RoboDK station: robodk_line_following_configuration_analysis.rdk

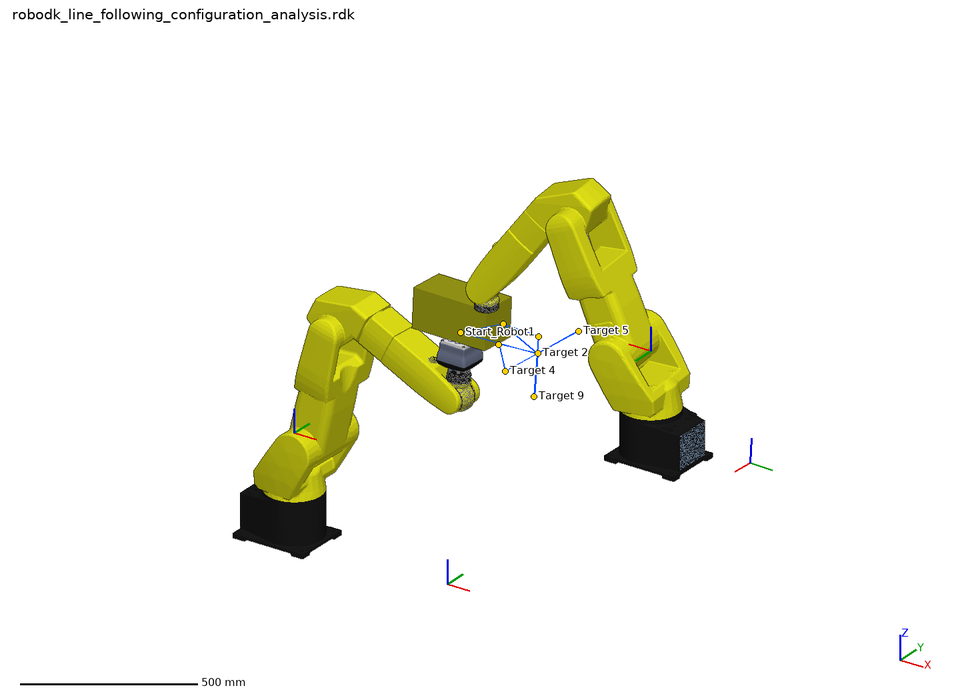
[picture v0: the station drawn from its stored meshes, robots at their saved joint values, targets as dots, program paths as lines]
Station Zavrsni_Line_Following_konfg (saved by RoboDK 5.9.4). Poses are relative to the parent item; angles as X-Y-Z fixed-axis rotations.
  - frame Pozicija 1 at (0, 0, 0) mm
    - frame Robot2 at (1093.21, 1000, 570) mm
      - robot Robot1: 6 axes
          modified DH rows (alpha deg, a mm, theta deg, d mm): 0, 0, 0, 330; -90, 75, -90, 0; 0, 400, 0, 0; -90, 75, 0, 410; 90, 0, 0, 0; -90, 0, 0, 80
          base shift (0, 0, -330) mm
          joint limits [-170, -60, -70, -190, -115, -400] to [170, 140, 170, 190, 115, 400]; home [0, 0, 0, 0, 0, 0]; saved at [-1.125, 13.477, -25.633, 3.463, 114.965, -89.87]
        - frame Kocka_Frame at (0, 1000, 0) mm
          - target Start_Robot2 (Cartesian target) at (63.45, -874.36, 243.45) mm, rotated rx 176.87 ry 0.69 rz -90 deg; joints [6.118, 22.277, -53.703, 0.008, -36.284, -5.881] of Robot2
          - target Kut_2 (Cartesian target) at (63.45, -1124.36, 243.45) mm, rotated rx 176.87 ry 0 rz -90 deg; joints [4.228, 52.378, -32.499, 0.062, -56.803, -4.056] of Robot2
          - target Kut_3 (Cartesian target) at (-60.55, -1124.36, 243.45) mm, rotated rx 176.87 ry 0 rz -90 deg; joints [-4.893, 52.997, -32.992, -0.071, -56.31, 5.138] of Robot2
          - target Kut_4 (Cartesian target) at (-60.55, -874.35, 243.45) mm, rotated rx 176.87 ry 0.69 rz -90.24 deg; joints [-7.279, 23.195, -54.517, 0, -35.483, 7.279] of Robot2
          - target Line_001 (Cartesian target) at (63.45, -874.36, 243.45) mm, rotated rx 176.87 ry 0.69 rz -90 deg; joints [-1.125, 13.477, -25.633, 3.463, 114.965, -89.87] of Robot2
          - target Line_002 (Cartesian target) at (63.45, -876.88, 243.45) mm, rotated rx 176.87 ry 0.69 rz -90 deg; joints [-1.125, 13.477, -25.633, 3.463, 114.965, -89.87] of Robot2
          - target Line_003 (Cartesian target) at (63.45, -879.41, 243.45) mm, rotated rx 176.87 ry 0.69 rz -90 deg; joints [-1.125, 13.477, -25.633, 3.463, 114.965, -89.87] of Robot2
          - target Line_004 (Cartesian target) at (63.45, -881.93, 243.45) mm, rotated rx 176.87 ry 0.69 rz -90 deg; joints [-1.125, 13.477, -25.633, 3.463, 114.965, -89.87] of Robot2
          - target Line_005 (Cartesian target) at (63.45, -884.46, 243.45) mm, rotated rx 176.87 ry 0.69 rz -90 deg; joints [-1.125, 13.477, -25.633, 3.463, 114.965, -89.87] of Robot2
          - target Line_006 (Cartesian target) at (63.45, -886.98, 243.45) mm, rotated rx 176.87 ry 0.69 rz -90 deg; joints [-1.125, 13.477, -25.633, 3.463, 114.965, -89.87] of Robot2
          - target Line_007 (Cartesian target) at (63.45, -889.51, 243.45) mm, rotated rx 176.87 ry 0.69 rz -90 deg; joints [-1.125, 13.477, -25.633, 3.463, 114.965, -89.87] of Robot2
          - target Line_008 (Cartesian target) at (63.45, -892.03, 243.45) mm, rotated rx 176.87 ry 0.69 rz -90 deg; joints [-1.125, 13.477, -25.633, 3.463, 114.965, -89.87] of Robot2
          - target Line_009 (Cartesian target) at (63.45, -894.56, 243.45) mm, rotated rx 176.87 ry 0.69 rz -90 deg; joints [-1.125, 13.477, -25.633, 3.463, 114.965, -89.87] of Robot2
          - target Line_010 (Cartesian target) at (63.45, -897.08, 243.45) mm, rotated rx 176.87 ry 0.69 rz -90 deg; joints [-1.125, 13.477, -25.633, 3.463, 114.965, -89.87] of Robot2
          - target Line_011 (Cartesian target) at (63.45, -899.61, 243.45) mm, rotated rx 176.87 ry 0.69 rz -90 deg; joints [-1.125, 13.477, -25.633, 3.463, 114.965, -89.87] of Robot2
          - target Line_012 (Cartesian target) at (63.45, -902.13, 243.45) mm, rotated rx 176.87 ry 0.69 rz -90 deg; joints [-1.125, 13.477, -25.633, 3.463, 114.965, -89.87] of Robot2
          - target Line_013 (Cartesian target) at (63.45, -904.66, 243.45) mm, rotated rx 176.87 ry 0.69 rz -90 deg; joints [-1.125, 13.477, -25.633, 3.463, 114.965, -89.87] of Robot2
          - target Line_014 (Cartesian target) at (63.45, -907.18, 243.45) mm, rotated rx 176.87 ry 0.69 rz -90 deg; joints [-1.125, 13.477, -25.633, 3.463, 114.965, -89.87] of Robot2
          - target Line_015 (Cartesian target) at (63.45, -909.71, 243.45) mm, rotated rx 176.87 ry 0.69 rz -90 deg; joints [-1.125, 13.477, -25.633, 3.463, 114.965, -89.87] of Robot2
          - target Line_016 (Cartesian target) at (63.45, -912.23, 243.45) mm, rotated rx 176.87 ry 0.69 rz -90 deg; joints [-1.125, 13.477, -25.633, 3.463, 114.965, -89.87] of Robot2
          - target Line_017 (Cartesian target) at (63.45, -914.76, 243.45) mm, rotated rx 176.87 ry 0.69 rz -90 deg; joints [-1.125, 13.477, -25.633, 3.463, 114.965, -89.87] of Robot2
          - target Line_018 (Cartesian target) at (63.45, -917.28, 243.45) mm, rotated rx 176.87 ry 0.69 rz -90 deg; joints [-1.125, 13.477, -25.633, 3.463, 114.965, -89.87] of Robot2
          - target Line_019 (Cartesian target) at (63.45, -919.81, 243.45) mm, rotated rx 176.87 ry 0.69 rz -90 deg; joints [-1.125, 13.477, -25.633, 3.463, 114.965, -89.87] of Robot2
          - target Line_020 (Cartesian target) at (63.45, -922.33, 243.45) mm, rotated rx 176.87 ry 0.69 rz -90 deg; joints [-1.125, 13.477, -25.633, 3.463, 114.965, -89.87] of Robot2
          - target Line_021 (Cartesian target) at (63.45, -924.86, 243.45) mm, rotated rx 176.87 ry 0.69 rz -90 deg; joints [-1.125, 13.477, -25.633, 3.463, 114.965, -89.87] of Robot2
          - target Line_022 (Cartesian target) at (63.45, -927.39, 243.45) mm, rotated rx 176.87 ry 0.69 rz -90 deg; joints [-1.125, 13.477, -25.633, 3.463, 114.965, -89.87] of Robot2
          - target Line_023 (Cartesian target) at (63.45, -929.91, 243.45) mm, rotated rx 176.87 ry 0.69 rz -90 deg; joints [-1.125, 13.477, -25.633, 3.463, 114.965, -89.87] of Robot2
          - target Line_024 (Cartesian target) at (63.45, -932.44, 243.45) mm, rotated rx 176.87 ry 0.69 rz -90 deg; joints [-1.125, 13.477, -25.633, 3.463, 114.965, -89.87] of Robot2
          - target Line_025 (Cartesian target) at (63.45, -934.96, 243.45) mm, rotated rx 176.87 ry 0.69 rz -90 deg; joints [-1.125, 13.477, -25.633, 3.463, 114.965, -89.87] of Robot2
          - target Line_026 (Cartesian target) at (63.45, -937.49, 243.45) mm, rotated rx 176.87 ry 0.69 rz -90 deg; joints [-1.125, 13.477, -25.633, 3.463, 114.965, -89.87] of Robot2
          - target Line_027 (Cartesian target) at (63.45, -940.01, 243.45) mm, rotated rx 176.87 ry 0.69 rz -90 deg; joints [-1.125, 13.477, -25.633, 3.463, 114.965, -89.87] of Robot2
          - target Line_028 (Cartesian target) at (63.45, -942.54, 243.45) mm, rotated rx 176.87 ry 0.69 rz -90 deg; joints [-1.125, 13.477, -25.633, 3.463, 114.965, -89.87] of Robot2
          - target Line_029 (Cartesian target) at (63.45, -945.06, 243.45) mm, rotated rx 176.87 ry 0.69 rz -90 deg; joints [-1.125, 13.477, -25.633, 3.463, 114.965, -89.87] of Robot2
          - target Line_030 (Cartesian target) at (63.45, -947.59, 243.45) mm, rotated rx 176.87 ry 0.69 rz -90 deg; joints [-1.125, 13.477, -25.633, 3.463, 114.965, -89.87] of Robot2
          - target Line_031 (Cartesian target) at (63.45, -950.11, 243.45) mm, rotated rx 176.87 ry 0.69 rz -90 deg; joints [-1.125, 13.477, -25.633, 3.463, 114.965, -89.87] of Robot2
          - target Line_032 (Cartesian target) at (63.45, -952.64, 243.45) mm, rotated rx 176.87 ry 0.69 rz -90 deg; joints [-1.125, 13.477, -25.633, 3.463, 114.965, -89.87] of Robot2
          - target Line_033 (Cartesian target) at (63.45, -955.16, 243.45) mm, rotated rx 176.87 ry 0.69 rz -90 deg; joints [-1.125, 13.477, -25.633, 3.463, 114.965, -89.87] of Robot2
          - target Line_034 (Cartesian target) at (63.45, -957.69, 243.45) mm, rotated rx 176.87 ry 0.69 rz -90 deg; joints [-1.125, 13.477, -25.633, 3.463, 114.965, -89.87] of Robot2
          - target Line_035 (Cartesian target) at (63.45, -960.21, 243.45) mm, rotated rx 176.87 ry 0.69 rz -90 deg; joints [-1.125, 13.477, -25.633, 3.463, 114.965, -89.87] of Robot2
          - target Line_036 (Cartesian target) at (63.45, -962.74, 243.45) mm, rotated rx 176.87 ry 0.69 rz -90 deg; joints [-1.125, 13.477, -25.633, 3.463, 114.965, -89.87] of Robot2
          - target Line_037 (Cartesian target) at (63.45, -965.26, 243.45) mm, rotated rx 176.87 ry 0.69 rz -90 deg; joints [-1.125, 13.477, -25.633, 3.463, 114.965, -89.87] of Robot2
          - target Line_038 (Cartesian target) at (63.45, -967.79, 243.45) mm, rotated rx 176.87 ry 0.69 rz -90 deg; joints [-1.125, 13.477, -25.633, 3.463, 114.965, -89.87] of Robot2
          - target Line_039 (Cartesian target) at (63.45, -970.31, 243.45) mm, rotated rx 176.87 ry 0.69 rz -90 deg; joints [-1.125, 13.477, -25.633, 3.463, 114.965, -89.87] of Robot2
          - target Line_040 (Cartesian target) at (63.45, -972.84, 243.45) mm, rotated rx 176.87 ry 0.69 rz -90 deg; joints [-1.125, 13.477, -25.633, 3.463, 114.965, -89.87] of Robot2
          - target Line_041 (Cartesian target) at (63.45, -975.37, 243.45) mm, rotated rx 176.87 ry 0.69 rz -90 deg; joints [-1.125, 13.477, -25.633, 3.463, 114.965, -89.87] of Robot2
          - target Line_042 (Cartesian target) at (63.45, -977.89, 243.45) mm, rotated rx 176.87 ry 0.69 rz -90 deg; joints [-1.125, 13.477, -25.633, 3.463, 114.965, -89.87] of Robot2
          - target Line_043 (Cartesian target) at (63.45, -980.42, 243.45) mm, rotated rx 176.87 ry 0.69 rz -90 deg; joints [-1.125, 13.477, -25.633, 3.463, 114.965, -89.87] of Robot2
          - target Line_044 (Cartesian target) at (63.45, -982.94, 243.45) mm, rotated rx 176.87 ry 0.69 rz -90 deg; joints [-1.125, 13.477, -25.633, 3.463, 114.965, -89.87] of Robot2
          - target Line_045 (Cartesian target) at (63.45, -985.47, 243.45) mm, rotated rx 176.87 ry 0.69 rz -90 deg; joints [-1.125, 13.477, -25.633, 3.463, 114.965, -89.87] of Robot2
          - target Line_046 (Cartesian target) at (63.45, -987.99, 243.45) mm, rotated rx 176.87 ry 0.69 rz -90 deg; joints [-1.125, 13.477, -25.633, 3.463, 114.965, -89.87] of Robot2
          - target Line_047 (Cartesian target) at (63.45, -990.52, 243.45) mm, rotated rx 176.87 ry 0.69 rz -90 deg; joints [-1.125, 13.477, -25.633, 3.463, 114.965, -89.87] of Robot2
          - target Line_048 (Cartesian target) at (63.45, -993.04, 243.45) mm, rotated rx 176.87 ry 0.69 rz -90 deg; joints [-1.125, 13.477, -25.633, 3.463, 114.965, -89.87] of Robot2
          - target Line_049 (Cartesian target) at (63.45, -995.57, 243.45) mm, rotated rx 176.87 ry 0.69 rz -90 deg; joints [-1.125, 13.477, -25.633, 3.463, 114.965, -89.87] of Robot2
          - target Line_050 (Cartesian target) at (63.45, -998.09, 243.45) mm, rotated rx 176.87 ry 0.69 rz -90 deg; joints [-1.125, 13.477, -25.633, 3.463, 114.965, -89.87] of Robot2
          - target Line_051 (Cartesian target) at (63.45, -1000.62, 243.45) mm, rotated rx 176.87 ry 0.69 rz -90 deg; joints [-1.125, 13.477, -25.633, 3.463, 114.965, -89.87] of Robot2
          - target Line_052 (Cartesian target) at (63.45, -1003.14, 243.45) mm, rotated rx 176.87 ry 0.69 rz -90 deg; joints [-1.125, 13.477, -25.633, 3.463, 114.965, -89.87] of Robot2
          - target Line_053 (Cartesian target) at (63.45, -1005.67, 243.45) mm, rotated rx 176.87 ry 0.69 rz -90 deg; joints [-1.125, 13.477, -25.633, 3.463, 114.965, -89.87] of Robot2
          - target Line_054 (Cartesian target) at (63.45, -1008.19, 243.45) mm, rotated rx 176.87 ry 0.69 rz -90 deg; joints [-1.125, 13.477, -25.633, 3.463, 114.965, -89.87] of Robot2
          - target Line_055 (Cartesian target) at (63.45, -1010.72, 243.45) mm, rotated rx 176.87 ry 0.69 rz -90 deg; joints [-1.125, 13.477, -25.633, 3.463, 114.965, -89.87] of Robot2
          - target Line_056 (Cartesian target) at (63.45, -1013.24, 243.45) mm, rotated rx 176.87 ry 0.69 rz -90 deg; joints [-1.125, 13.477, -25.633, 3.463, 114.965, -89.87] of Robot2
          - target Line_057 (Cartesian target) at (63.45, -1015.77, 243.45) mm, rotated rx 176.87 ry 0.69 rz -90 deg; joints [-1.125, 13.477, -25.633, 3.463, 114.965, -89.87] of Robot2
          - target Line_058 (Cartesian target) at (63.45, -1018.29, 243.45) mm, rotated rx 176.87 ry 0.69 rz -90 deg; joints [-1.125, 13.477, -25.633, 3.463, 114.965, -89.87] of Robot2
          - target Line_059 (Cartesian target) at (63.45, -1020.82, 243.45) mm, rotated rx 176.87 ry 0.69 rz -90 deg; joints [-1.125, 13.477, -25.633, 3.463, 114.965, -89.87] of Robot2
          - target Line_060 (Cartesian target) at (63.45, -1023.34, 243.45) mm, rotated rx 176.87 ry 0.69 rz -90 deg; joints [-1.125, 13.477, -25.633, 3.463, 114.965, -89.87] of Robot2
          - target Line_061 (Cartesian target) at (63.45, -1025.87, 243.45) mm, rotated rx 176.87 ry 0.69 rz -90 deg; joints [-1.125, 13.477, -25.633, 3.463, 114.965, -89.87] of Robot2
          - target Line_062 (Cartesian target) at (63.45, -1028.4, 243.45) mm, rotated rx 176.87 ry 0.69 rz -90 deg; joints [-1.125, 13.477, -25.633, 3.463, 114.965, -89.87] of Robot2
          - target Line_063 (Cartesian target) at (63.45, -1030.92, 243.45) mm, rotated rx 176.87 ry 0.69 rz -90 deg; joints [-1.125, 13.477, -25.633, 3.463, 114.965, -89.87] of Robot2
          - target Line_064 (Cartesian target) at (63.45, -1033.45, 243.45) mm, rotated rx 176.87 ry 0.69 rz -90 deg; joints [-1.125, 13.477, -25.633, 3.463, 114.965, -89.87] of Robot2
          - target Line_065 (Cartesian target) at (63.45, -1035.97, 243.45) mm, rotated rx 176.87 ry 0.69 rz -90 deg; joints [-1.125, 13.477, -25.633, 3.463, 114.965, -89.87] of Robot2
          - target Line_066 (Cartesian target) at (63.45, -1038.5, 243.45) mm, rotated rx 176.87 ry 0.69 rz -90 deg; joints [-1.125, 13.477, -25.633, 3.463, 114.965, -89.87] of Robot2
          - target Line_067 (Cartesian target) at (63.45, -1041.02, 243.45) mm, rotated rx 176.87 ry 0.69 rz -90 deg; joints [-1.125, 13.477, -25.633, 3.463, 114.965, -89.87] of Robot2
          - target Line_068 (Cartesian target) at (63.45, -1043.55, 243.45) mm, rotated rx 176.87 ry 0.69 rz -90 deg; joints [-1.125, 13.477, -25.633, 3.463, 114.965, -89.87] of Robot2
          - target Line_069 (Cartesian target) at (63.45, -1046.07, 243.45) mm, rotated rx 176.87 ry 0.69 rz -90 deg; joints [-1.125, 13.477, -25.633, 3.463, 114.965, -89.87] of Robot2
          - target Line_070 (Cartesian target) at (63.45, -1048.6, 243.45) mm, rotated rx 176.87 ry 0.69 rz -90 deg; joints [-1.125, 13.477, -25.633, 3.463, 114.965, -89.87] of Robot2
          - target Line_071 (Cartesian target) at (63.45, -1051.12, 243.45) mm, rotated rx 176.87 ry 0.69 rz -90 deg; joints [-1.125, 13.477, -25.633, 3.463, 114.965, -89.87] of Robot2
          - target Line_072 (Cartesian target) at (63.45, -1053.65, 243.45) mm, rotated rx 176.87 ry 0.69 rz -90 deg; joints [-1.125, 13.477, -25.633, 3.463, 114.965, -89.87] of Robot2
          - target Line_073 (Cartesian target) at (63.45, -1056.17, 243.45) mm, rotated rx 176.87 ry 0.69 rz -90 deg; joints [-1.125, 13.477, -25.633, 3.463, 114.965, -89.87] of Robot2
          - target Line_074 (Cartesian target) at (63.45, -1058.7, 243.45) mm, rotated rx 176.87 ry 0.69 rz -90 deg; joints [-1.125, 13.477, -25.633, 3.463, 114.965, -89.87] of Robot2
          - target Line_075 (Cartesian target) at (63.45, -1061.22, 243.45) mm, rotated rx 176.87 ry 0.69 rz -90 deg; joints [-1.125, 13.477, -25.633, 3.463, 114.965, -89.87] of Robot2
          - target Line_076 (Cartesian target) at (63.45, -1063.75, 243.45) mm, rotated rx 176.87 ry 0.69 rz -90 deg; joints [-1.125, 13.477, -25.633, 3.463, 114.965, -89.87] of Robot2
          - target Line_077 (Cartesian target) at (63.45, -1066.27, 243.45) mm, rotated rx 176.87 ry 0.69 rz -90 deg; joints [-1.125, 13.477, -25.633, 3.463, 114.965, -89.87] of Robot2
          - target Line_078 (Cartesian target) at (63.45, -1068.8, 243.45) mm, rotated rx 176.87 ry 0.69 rz -90 deg; joints [-1.125, 13.477, -25.633, 3.463, 114.965, -89.87] of Robot2
          - target Line_079 (Cartesian target) at (63.45, -1071.32, 243.45) mm, rotated rx 176.87 ry 0.69 rz -90 deg; joints [-1.125, 13.477, -25.633, 3.463, 114.965, -89.87] of Robot2
          - target Line_080 (Cartesian target) at (63.45, -1073.85, 243.45) mm, rotated rx 176.87 ry 0.69 rz -90 deg; joints [-1.125, 13.477, -25.633, 3.463, 114.965, -89.87] of Robot2
          - target Line_081 (Cartesian target) at (63.45, -1076.38, 243.45) mm, rotated rx 176.87 ry 0.69 rz -90 deg; joints [-1.125, 13.477, -25.633, 3.463, 114.965, -89.87] of Robot2
          - target Line_082 (Cartesian target) at (63.45, -1078.9, 243.45) mm, rotated rx 176.87 ry 0.69 rz -90 deg; joints [-1.125, 13.477, -25.633, 3.463, 114.965, -89.87] of Robot2
          - target Line_083 (Cartesian target) at (63.45, -1081.43, 243.45) mm, rotated rx 176.87 ry 0.69 rz -90 deg; joints [-1.125, 13.477, -25.633, 3.463, 114.965, -89.87] of Robot2
          - target Line_084 (Cartesian target) at (63.45, -1083.95, 243.45) mm, rotated rx 176.87 ry 0.69 rz -90 deg; joints [-1.125, 13.477, -25.633, 3.463, 114.965, -89.87] of Robot2
          - target Line_085 (Cartesian target) at (63.45, -1086.48, 243.45) mm, rotated rx 176.87 ry 0.69 rz -90 deg; joints [-1.125, 13.477, -25.633, 3.463, 114.965, -89.87] of Robot2
          - target Line_086 (Cartesian target) at (63.45, -1089, 243.45) mm, rotated rx 176.87 ry 0.69 rz -90 deg; joints [-1.125, 13.477, -25.633, 3.463, 114.965, -89.87] of Robot2
          - target Line_087 (Cartesian target) at (63.45, -1091.53, 243.45) mm, rotated rx 176.87 ry 0.69 rz -90 deg; joints [-1.125, 13.477, -25.633, 3.463, 114.965, -89.87] of Robot2
          - target Line_088 (Cartesian target) at (63.45, -1094.05, 243.45) mm, rotated rx 176.87 ry 0.69 rz -90 deg; joints [-1.125, 13.477, -25.633, 3.463, 114.965, -89.87] of Robot2
          - target Line_089 (Cartesian target) at (63.45, -1096.58, 243.45) mm, rotated rx 176.87 ry 0.69 rz -90 deg; joints [-1.125, 13.477, -25.633, 3.463, 114.965, -89.87] of Robot2
          - target Line_090 (Cartesian target) at (63.45, -1099.1, 243.45) mm, rotated rx 176.87 ry 0.69 rz -90 deg; joints [-1.125, 13.477, -25.633, 3.463, 114.965, -89.87] of Robot2
          - target Line_091 (Cartesian target) at (63.45, -1101.63, 243.45) mm, rotated rx 176.87 ry 0.69 rz -90 deg; joints [-1.125, 13.477, -25.633, 3.463, 114.965, -89.87] of Robot2
          - target Line_092 (Cartesian target) at (63.45, -1104.15, 243.45) mm, rotated rx 176.87 ry 0.69 rz -90 deg; joints [-1.125, 13.477, -25.633, 3.463, 114.965, -89.87] of Robot2
          - target Line_093 (Cartesian target) at (63.45, -1106.68, 243.45) mm, rotated rx 176.87 ry 0.69 rz -90 deg; joints [-1.125, 13.477, -25.633, 3.463, 114.965, -89.87] of Robot2
          - target Line_094 (Cartesian target) at (63.45, -1109.2, 243.45) mm, rotated rx 176.87 ry 0.69 rz -90 deg; joints [-1.125, 13.477, -25.633, 3.463, 114.965, -89.87] of Robot2
          - target Line_095 (Cartesian target) at (63.45, -1111.73, 243.45) mm, rotated rx 176.87 ry 0.69 rz -90 deg; joints [-1.125, 13.477, -25.633, 3.463, 114.965, -89.87] of Robot2
          - target Line_096 (Cartesian target) at (63.45, -1114.25, 243.45) mm, rotated rx 176.87 ry 0.69 rz -90 deg; joints [-1.125, 13.477, -25.633, 3.463, 114.965, -89.87] of Robot2
          - target Line_097 (Cartesian target) at (63.45, -1116.78, 243.45) mm, rotated rx 176.87 ry 0.69 rz -90 deg; joints [-1.125, 13.477, -25.633, 3.463, 114.965, -89.87] of Robot2
          - target Line_098 (Cartesian target) at (63.45, -1119.3, 243.45) mm, rotated rx 176.87 ry 0.69 rz -90 deg; joints [-1.125, 13.477, -25.633, 3.463, 114.965, -89.87] of Robot2
          - target Line_099 (Cartesian target) at (63.45, -1121.83, 243.45) mm, rotated rx 176.87 ry 0.69 rz -90 deg; joints [-1.125, 13.477, -25.633, 3.463, 114.965, -89.87] of Robot2
          - target Line_100 (Cartesian target) at (63.45, -1124.36, 243.45) mm, rotated rx 176.87 ry 0.69 rz -90 deg; joints [-1.125, 13.477, -25.633, 3.463, 114.965, -89.87] of Robot2
          - target Line_101 (Cartesian target) at (63.45, -1124.36, 243.45) mm, rotated rx 176.87 ry 0 rz -90 deg; joints [-1.125, 13.477, -25.633, 3.463, 114.965, -89.87] of Robot2
          - target Line_102 (Cartesian target) at (62.2, -1124.36, 243.45) mm, rotated rx 176.87 ry 0 rz -90 deg; joints [-1.125, 13.477, -25.633, 3.463, 114.965, -89.87] of Robot2
          - target Line_103 (Cartesian target) at (60.94, -1124.36, 243.45) mm, rotated rx 176.87 ry 0 rz -90 deg; joints [-1.125, 13.477, -25.633, 3.463, 114.965, -89.87] of Robot2
          - target Line_104 (Cartesian target) at (59.69, -1124.36, 243.45) mm, rotated rx 176.87 ry 0 rz -90 deg; joints [-1.125, 13.477, -25.633, 3.463, 114.965, -89.87] of Robot2
          - target Line_105 (Cartesian target) at (58.44, -1124.36, 243.45) mm, rotated rx 176.87 ry 0 rz -90 deg; joints [-1.125, 13.477, -25.633, 3.463, 114.965, -89.87] of Robot2
          - target Line_106 (Cartesian target) at (57.19, -1124.36, 243.45) mm, rotated rx 176.87 ry 0 rz -90 deg; joints [-1.125, 13.477, -25.633, 3.463, 114.965, -89.87] of Robot2
          - target Line_107 (Cartesian target) at (55.93, -1124.36, 243.45) mm, rotated rx 176.87 ry 0 rz -90 deg; joints [-1.125, 13.477, -25.633, 3.463, 114.965, -89.87] of Robot2
          - target Line_108 (Cartesian target) at (54.68, -1124.36, 243.45) mm, rotated rx 176.87 ry 0 rz -90 deg; joints [-1.125, 13.477, -25.633, 3.463, 114.965, -89.87] of Robot2
          - target Line_109 (Cartesian target) at (53.43, -1124.36, 243.45) mm, rotated rx 176.87 ry 0 rz -90 deg; joints [-1.125, 13.477, -25.633, 3.463, 114.965, -89.87] of Robot2
          - target Line_110 (Cartesian target) at (52.18, -1124.36, 243.45) mm, rotated rx 176.87 ry 0 rz -90 deg; joints [-1.125, 13.477, -25.633, 3.463, 114.965, -89.87] of Robot2
          - target Line_111 (Cartesian target) at (50.92, -1124.36, 243.45) mm, rotated rx 176.87 ry 0 rz -90 deg; joints [-1.125, 13.477, -25.633, 3.463, 114.965, -89.87] of Robot2
          - target Line_112 (Cartesian target) at (49.67, -1124.36, 243.45) mm, rotated rx 176.87 ry 0 rz -90 deg; joints [-1.125, 13.477, -25.633, 3.463, 114.965, -89.87] of Robot2
          - target Line_113 (Cartesian target) at (48.42, -1124.36, 243.45) mm, rotated rx 176.87 ry 0 rz -90 deg; joints [-1.125, 13.477, -25.633, 3.463, 114.965, -89.87] of Robot2
          - target Line_114 (Cartesian target) at (47.17, -1124.36, 243.45) mm, rotated rx 176.87 ry 0 rz -90 deg; joints [-1.125, 13.477, -25.633, 3.463, 114.965, -89.87] of Robot2
          - target Line_115 (Cartesian target) at (45.91, -1124.36, 243.45) mm, rotated rx 176.87 ry 0 rz -90 deg; joints [-1.125, 13.477, -25.633, 3.463, 114.965, -89.87] of Robot2
          - target Line_116 (Cartesian target) at (44.66, -1124.36, 243.45) mm, rotated rx 176.87 ry 0 rz -90 deg; joints [-1.125, 13.477, -25.633, 3.463, 114.965, -89.87] of Robot2
          - target Line_117 (Cartesian target) at (43.41, -1124.36, 243.45) mm, rotated rx 176.87 ry 0 rz -90 deg; joints [-1.125, 13.477, -25.633, 3.463, 114.965, -89.87] of Robot2
          - target Line_118 (Cartesian target) at (42.16, -1124.36, 243.45) mm, rotated rx 176.87 ry 0 rz -90 deg; joints [-1.125, 13.477, -25.633, 3.463, 114.965, -89.87] of Robot2
          - target Line_119 (Cartesian target) at (40.9, -1124.36, 243.45) mm, rotated rx 176.87 ry 0 rz -90 deg; joints [-1.125, 13.477, -25.633, 3.463, 114.965, -89.87] of Robot2
          - target Line_120 (Cartesian target) at (39.65, -1124.36, 243.45) mm, rotated rx 176.87 ry 0 rz -90 deg; joints [-1.125, 13.477, -25.633, 3.463, 114.965, -89.87] of Robot2
          - target Line_121 (Cartesian target) at (38.4, -1124.36, 243.45) mm, rotated rx 176.87 ry 0 rz -90 deg; joints [-1.125, 13.477, -25.633, 3.463, 114.965, -89.87] of Robot2
          - target Line_122 (Cartesian target) at (37.14, -1124.36, 243.45) mm, rotated rx 176.87 ry 0 rz -90 deg; joints [-1.125, 13.477, -25.633, 3.463, 114.965, -89.87] of Robot2
          - target Line_123 (Cartesian target) at (35.89, -1124.36, 243.45) mm, rotated rx 176.87 ry 0 rz -90 deg; joints [-1.125, 13.477, -25.633, 3.463, 114.965, -89.87] of Robot2
          - target Line_124 (Cartesian target) at (34.64, -1124.36, 243.45) mm, rotated rx 176.87 ry 0 rz -90 deg; joints [-1.125, 13.477, -25.633, 3.463, 114.965, -89.87] of Robot2
          - target Line_125 (Cartesian target) at (33.39, -1124.36, 243.45) mm, rotated rx 176.87 ry 0 rz -90 deg; joints [-1.125, 13.477, -25.633, 3.463, 114.965, -89.87] of Robot2
          - target Line_126 (Cartesian target) at (32.13, -1124.36, 243.45) mm, rotated rx 176.87 ry 0 rz -90 deg; joints [-1.125, 13.477, -25.633, 3.463, 114.965, -89.87] of Robot2
          - target Line_127 (Cartesian target) at (30.88, -1124.36, 243.45) mm, rotated rx 176.87 ry 0 rz -90 deg; joints [-1.125, 13.477, -25.633, 3.463, 114.965, -89.87] of Robot2
          - target Line_128 (Cartesian target) at (29.63, -1124.36, 243.45) mm, rotated rx 176.87 ry 0 rz -90 deg; joints [-1.125, 13.477, -25.633, 3.463, 114.965, -89.87] of Robot2
          - target Line_129 (Cartesian target) at (28.38, -1124.36, 243.45) mm, rotated rx 176.87 ry 0 rz -90 deg; joints [-1.125, 13.477, -25.633, 3.463, 114.965, -89.87] of Robot2
          - target Line_130 (Cartesian target) at (27.12, -1124.36, 243.45) mm, rotated rx 176.87 ry 0 rz -90 deg; joints [-1.125, 13.477, -25.633, 3.463, 114.965, -89.87] of Robot2
          - target Line_131 (Cartesian target) at (25.87, -1124.36, 243.45) mm, rotated rx 176.87 ry 0 rz -90 deg; joints [-1.125, 13.477, -25.633, 3.463, 114.965, -89.87] of Robot2
          - target Line_132 (Cartesian target) at (24.62, -1124.36, 243.45) mm, rotated rx 176.87 ry 0 rz -90 deg; joints [-1.125, 13.477, -25.633, 3.463, 114.965, -89.87] of Robot2
          - target Line_133 (Cartesian target) at (23.37, -1124.36, 243.45) mm, rotated rx 176.87 ry 0 rz -90 deg; joints [-1.125, 13.477, -25.633, 3.463, 114.965, -89.87] of Robot2
          - target Line_134 (Cartesian target) at (22.11, -1124.36, 243.45) mm, rotated rx 176.87 ry 0 rz -90 deg; joints [-1.125, 13.477, -25.633, 3.463, 114.965, -89.87] of Robot2
          - target Line_135 (Cartesian target) at (20.86, -1124.36, 243.45) mm, rotated rx 176.87 ry 0 rz -90 deg; joints [-1.125, 13.477, -25.633, 3.463, 114.965, -89.87] of Robot2
          - target Line_136 (Cartesian target) at (19.61, -1124.36, 243.45) mm, rotated rx 176.87 ry 0 rz -90 deg; joints [-1.125, 13.477, -25.633, 3.463, 114.965, -89.87] of Robot2
          - target Line_137 (Cartesian target) at (18.36, -1124.36, 243.45) mm, rotated rx 176.87 ry 0 rz -90 deg; joints [-1.125, 13.477, -25.633, 3.463, 114.965, -89.87] of Robot2
          - target Line_138 (Cartesian target) at (17.1, -1124.36, 243.45) mm, rotated rx 176.87 ry 0 rz -90 deg; joints [-1.125, 13.477, -25.633, 3.463, 114.965, -89.87] of Robot2
          - target Line_139 (Cartesian target) at (15.85, -1124.36, 243.45) mm, rotated rx 176.87 ry 0 rz -90 deg; joints [-1.125, 13.477, -25.633, 3.463, 114.965, -89.87] of Robot2
          - target Line_140 (Cartesian target) at (14.6, -1124.36, 243.45) mm, rotated rx 176.87 ry 0 rz -90 deg; joints [-1.125, 13.477, -25.633, 3.463, 114.965, -89.87] of Robot2
          - target Line_141 (Cartesian target) at (13.35, -1124.36, 243.45) mm, rotated rx 176.87 ry 0 rz -90 deg; joints [-1.125, 13.477, -25.633, 3.463, 114.965, -89.87] of Robot2
          - target Line_142 (Cartesian target) at (12.09, -1124.36, 243.45) mm, rotated rx 176.87 ry 0 rz -90 deg; joints [-1.125, 13.477, -25.633, 3.463, 114.965, -89.87] of Robot2
          - target Line_143 (Cartesian target) at (10.84, -1124.36, 243.45) mm, rotated rx 176.87 ry 0 rz -90 deg; joints [-1.125, 13.477, -25.633, 3.463, 114.965, -89.87] of Robot2
          - target Line_144 (Cartesian target) at (9.59, -1124.36, 243.45) mm, rotated rx 176.87 ry 0 rz -90 deg; joints [-1.125, 13.477, -25.633, 3.463, 114.965, -89.87] of Robot2
          - target Line_145 (Cartesian target) at (8.34, -1124.36, 243.45) mm, rotated rx 176.87 ry 0 rz -90 deg; joints [-1.125, 13.477, -25.633, 3.463, 114.965, -89.87] of Robot2
          - target Line_146 (Cartesian target) at (7.08, -1124.36, 243.45) mm, rotated rx 176.87 ry 0 rz -90 deg; joints [-1.125, 13.477, -25.633, 3.463, 114.965, -89.87] of Robot2
          - target Line_147 (Cartesian target) at (5.83, -1124.36, 243.45) mm, rotated rx 176.87 ry 0 rz -90 deg; joints [-1.125, 13.477, -25.633, 3.463, 114.965, -89.87] of Robot2
          - target Line_148 (Cartesian target) at (4.58, -1124.36, 243.45) mm, rotated rx 176.87 ry 0 rz -90 deg; joints [-1.125, 13.477, -25.633, 3.463, 114.965, -89.87] of Robot2
          - target Line_149 (Cartesian target) at (3.33, -1124.36, 243.45) mm, rotated rx 176.87 ry 0 rz -90 deg; joints [-1.125, 13.477, -25.633, 3.463, 114.965, -89.87] of Robot2
          - target Line_150 (Cartesian target) at (2.07, -1124.36, 243.45) mm, rotated rx 176.87 ry 0 rz -90 deg; joints [-1.125, 13.477, -25.633, 3.463, 114.965, -89.87] of Robot2
          - target Line_151 (Cartesian target) at (0.82, -1124.36, 243.45) mm, rotated rx 176.87 ry 0 rz -90 deg; joints [-1.125, 13.477, -25.633, 3.463, 114.965, -89.87] of Robot2
          - target Line_152 (Cartesian target) at (-0.43, -1124.36, 243.45) mm, rotated rx 176.87 ry 0 rz -90 deg; joints [-1.125, 13.477, -25.633, 3.463, 114.965, -89.87] of Robot2
          - target Line_153 (Cartesian target) at (-1.68, -1124.36, 243.45) mm, rotated rx 176.87 ry 0 rz -90 deg; joints [-1.125, 13.477, -25.633, 3.463, 114.965, -89.87] of Robot2
          - target Line_154 (Cartesian target) at (-2.94, -1124.36, 243.45) mm, rotated rx 176.87 ry 0 rz -90 deg; joints [-1.125, 13.477, -25.633, 3.463, 114.965, -89.87] of Robot2
          - target Line_155 (Cartesian target) at (-4.19, -1124.36, 243.45) mm, rotated rx 176.87 ry 0 rz -90 deg; joints [-1.125, 13.477, -25.633, 3.463, 114.965, -89.87] of Robot2
          - target Line_156 (Cartesian target) at (-5.44, -1124.36, 243.45) mm, rotated rx 176.87 ry 0 rz -90 deg; joints [-1.125, 13.477, -25.633, 3.463, 114.965, -89.87] of Robot2
          - target Line_157 (Cartesian target) at (-6.69, -1124.36, 243.45) mm, rotated rx 176.87 ry 0 rz -90 deg; joints [-1.125, 13.477, -25.633, 3.463, 114.965, -89.87] of Robot2
          - target Line_158 (Cartesian target) at (-7.95, -1124.36, 243.45) mm, rotated rx 176.87 ry 0 rz -90 deg; joints [-1.125, 13.477, -25.633, 3.463, 114.965, -89.87] of Robot2
          - target Line_159 (Cartesian target) at (-9.2, -1124.36, 243.45) mm, rotated rx 176.87 ry 0 rz -90 deg; joints [-1.125, 13.477, -25.633, 3.463, 114.965, -89.87] of Robot2
          - target Line_160 (Cartesian target) at (-10.45, -1124.36, 243.45) mm, rotated rx 176.87 ry 0 rz -90 deg; joints [-1.125, 13.477, -25.633, 3.463, 114.965, -89.87] of Robot2
          - target Line_161 (Cartesian target) at (-11.7, -1124.36, 243.45) mm, rotated rx 176.87 ry 0 rz -90 deg; joints [-1.125, 13.477, -25.633, 3.463, 114.965, -89.87] of Robot2
          - target Line_162 (Cartesian target) at (-12.96, -1124.36, 243.45) mm, rotated rx 176.87 ry 0 rz -90 deg; joints [-1.125, 13.477, -25.633, 3.463, 114.965, -89.87] of Robot2
          - target Line_163 (Cartesian target) at (-14.21, -1124.36, 243.45) mm, rotated rx 176.87 ry 0 rz -90 deg; joints [-1.125, 13.477, -25.633, 3.463, 114.965, -89.87] of Robot2
          - target Line_164 (Cartesian target) at (-15.46, -1124.36, 243.45) mm, rotated rx 176.87 ry 0 rz -90 deg; joints [-1.125, 13.477, -25.633, 3.463, 114.965, -89.87] of Robot2
          - target Line_165 (Cartesian target) at (-16.71, -1124.36, 243.45) mm, rotated rx 176.87 ry 0 rz -90 deg; joints [-1.125, 13.477, -25.633, 3.463, 114.965, -89.87] of Robot2
          - target Line_166 (Cartesian target) at (-17.97, -1124.36, 243.45) mm, rotated rx 176.87 ry 0 rz -90 deg; joints [-1.125, 13.477, -25.633, 3.463, 114.965, -89.87] of Robot2
          - target Line_167 (Cartesian target) at (-19.22, -1124.36, 243.45) mm, rotated rx 176.87 ry 0 rz -90 deg; joints [-1.125, 13.477, -25.633, 3.463, 114.965, -89.87] of Robot2
          - target Line_168 (Cartesian target) at (-20.47, -1124.36, 243.45) mm, rotated rx 176.87 ry 0 rz -90 deg; joints [-1.125, 13.477, -25.633, 3.463, 114.965, -89.87] of Robot2
          - target Line_169 (Cartesian target) at (-21.72, -1124.36, 243.45) mm, rotated rx 176.87 ry 0 rz -90 deg; joints [-1.125, 13.477, -25.633, 3.463, 114.965, -89.87] of Robot2
          - target Line_170 (Cartesian target) at (-22.98, -1124.36, 243.45) mm, rotated rx 176.87 ry 0 rz -90 deg; joints [-1.125, 13.477, -25.633, 3.463, 114.965, -89.87] of Robot2
          - target Line_171 (Cartesian target) at (-24.23, -1124.36, 243.45) mm, rotated rx 176.87 ry 0 rz -90 deg; joints [-1.125, 13.477, -25.633, 3.463, 114.965, -89.87] of Robot2
          - target Line_172 (Cartesian target) at (-25.48, -1124.36, 243.45) mm, rotated rx 176.87 ry 0 rz -90 deg; joints [-1.125, 13.477, -25.633, 3.463, 114.965, -89.87] of Robot2
          - target Line_173 (Cartesian target) at (-26.73, -1124.36, 243.45) mm, rotated rx 176.87 ry 0 rz -90 deg; joints [-1.125, 13.477, -25.633, 3.463, 114.965, -89.87] of Robot2
          - target Line_174 (Cartesian target) at (-27.99, -1124.36, 243.45) mm, rotated rx 176.87 ry 0 rz -90 deg; joints [-1.125, 13.477, -25.633, 3.463, 114.965, -89.87] of Robot2
          - target Line_175 (Cartesian target) at (-29.24, -1124.36, 243.45) mm, rotated rx 176.87 ry 0 rz -90 deg; joints [-1.125, 13.477, -25.633, 3.463, 114.965, -89.87] of Robot2
          - target Line_176 (Cartesian target) at (-30.49, -1124.36, 243.45) mm, rotated rx 176.87 ry 0 rz -90 deg; joints [-1.125, 13.477, -25.633, 3.463, 114.965, -89.87] of Robot2
          - target Line_177 (Cartesian target) at (-31.74, -1124.36, 243.45) mm, rotated rx 176.87 ry 0 rz -90 deg; joints [-1.125, 13.477, -25.633, 3.463, 114.965, -89.87] of Robot2
          - target Line_178 (Cartesian target) at (-33, -1124.36, 243.45) mm, rotated rx 176.87 ry 0 rz -90 deg; joints [-1.125, 13.477, -25.633, 3.463, 114.965, -89.87] of Robot2
          - target Line_179 (Cartesian target) at (-34.25, -1124.36, 243.45) mm, rotated rx 176.87 ry 0 rz -90 deg; joints [-1.125, 13.477, -25.633, 3.463, 114.965, -89.87] of Robot2
          - target Line_180 (Cartesian target) at (-35.5, -1124.36, 243.45) mm, rotated rx 176.87 ry 0 rz -90 deg; joints [-1.125, 13.477, -25.633, 3.463, 114.965, -89.87] of Robot2
          - target Line_181 (Cartesian target) at (-36.75, -1124.36, 243.45) mm, rotated rx 176.87 ry 0 rz -90 deg; joints [-1.125, 13.477, -25.633, 3.463, 114.965, -89.87] of Robot2
          - target Line_182 (Cartesian target) at (-38.01, -1124.36, 243.45) mm, rotated rx 176.87 ry 0 rz -90 deg; joints [-1.125, 13.477, -25.633, 3.463, 114.965, -89.87] of Robot2
          - target Line_183 (Cartesian target) at (-39.26, -1124.36, 243.45) mm, rotated rx 176.87 ry 0 rz -90 deg; joints [-1.125, 13.477, -25.633, 3.463, 114.965, -89.87] of Robot2
          - target Line_184 (Cartesian target) at (-40.51, -1124.36, 243.45) mm, rotated rx 176.87 ry 0 rz -90 deg; joints [-1.125, 13.477, -25.633, 3.463, 114.965, -89.87] of Robot2
          - target Line_185 (Cartesian target) at (-41.76, -1124.36, 243.45) mm, rotated rx 176.87 ry 0 rz -90 deg; joints [-1.125, 13.477, -25.633, 3.463, 114.965, -89.87] of Robot2
          - target Line_186 (Cartesian target) at (-43.02, -1124.36, 243.45) mm, rotated rx 176.87 ry 0 rz -90 deg; joints [-1.125, 13.477, -25.633, 3.463, 114.965, -89.87] of Robot2
          - target Line_187 (Cartesian target) at (-44.27, -1124.36, 243.45) mm, rotated rx 176.87 ry 0 rz -90 deg; joints [-1.125, 13.477, -25.633, 3.463, 114.965, -89.87] of Robot2
          - target Line_188 (Cartesian target) at (-45.52, -1124.36, 243.45) mm, rotated rx 176.87 ry 0 rz -90 deg; joints [-1.125, 13.477, -25.633, 3.463, 114.965, -89.87] of Robot2
          - target Line_189 (Cartesian target) at (-46.77, -1124.36, 243.45) mm, rotated rx 176.87 ry 0 rz -90 deg; joints [-1.125, 13.477, -25.633, 3.463, 114.965, -89.87] of Robot2
          - target Line_190 (Cartesian target) at (-48.03, -1124.36, 243.45) mm, rotated rx 176.87 ry 0 rz -90 deg; joints [-1.125, 13.477, -25.633, 3.463, 114.965, -89.87] of Robot2
          - target Line_191 (Cartesian target) at (-49.28, -1124.36, 243.45) mm, rotated rx 176.87 ry 0 rz -90 deg; joints [-1.125, 13.477, -25.633, 3.463, 114.965, -89.87] of Robot2
          - target Line_192 (Cartesian target) at (-50.53, -1124.36, 243.45) mm, rotated rx 176.87 ry 0 rz -90 deg; joints [-1.125, 13.477, -25.633, 3.463, 114.965, -89.87] of Robot2
          - target Line_193 (Cartesian target) at (-51.78, -1124.36, 243.45) mm, rotated rx 176.87 ry 0 rz -90 deg; joints [-1.125, 13.477, -25.633, 3.463, 114.965, -89.87] of Robot2
          - target Line_194 (Cartesian target) at (-53.04, -1124.36, 243.45) mm, rotated rx 176.87 ry 0 rz -90 deg; joints [-1.125, 13.477, -25.633, 3.463, 114.965, -89.87] of Robot2
          - target Line_195 (Cartesian target) at (-54.29, -1124.36, 243.45) mm, rotated rx 176.87 ry 0 rz -90 deg; joints [-1.125, 13.477, -25.633, 3.463, 114.965, -89.87] of Robot2
          - target Line_196 (Cartesian target) at (-55.54, -1124.36, 243.45) mm, rotated rx 176.87 ry 0 rz -90 deg; joints [-1.125, 13.477, -25.633, 3.463, 114.965, -89.87] of Robot2
          - target Line_197 (Cartesian target) at (-56.79, -1124.36, 243.45) mm, rotated rx 176.87 ry 0 rz -90 deg; joints [-1.125, 13.477, -25.633, 3.463, 114.965, -89.87] of Robot2
          - target Line_198 (Cartesian target) at (-58.05, -1124.36, 243.45) mm, rotated rx 176.87 ry 0 rz -90 deg; joints [-1.125, 13.477, -25.633, 3.463, 114.965, -89.87] of Robot2
          - target Line_199 (Cartesian target) at (-59.3, -1124.36, 243.45) mm, rotated rx 176.87 ry 0 rz -90 deg; joints [-1.125, 13.477, -25.633, 3.463, 114.965, -89.87] of Robot2
          - target Line_200 (Cartesian target) at (-60.55, -1124.36, 243.45) mm, rotated rx 176.87 ry 0 rz -90 deg; joints [-1.125, 13.477, -25.633, 3.463, 114.965, -89.87] of Robot2
          - target Line_201 (Cartesian target) at (-60.55, -1124.36, 243.45) mm, rotated rx 176.87 ry 0 rz -90 deg; joints [-1.125, 13.477, -25.633, 3.463, 114.965, -89.87] of Robot2
          - target Line_202 (Cartesian target) at (-60.55, -1121.83, 243.45) mm, rotated rx 176.87 ry 0 rz -90 deg; joints [-1.125, 13.477, -25.633, 3.463, 114.965, -89.87] of Robot2
          - target Line_203 (Cartesian target) at (-60.55, -1119.3, 243.45) mm, rotated rx 176.87 ry 0 rz -90 deg; joints [-1.125, 13.477, -25.633, 3.463, 114.965, -89.87] of Robot2
          - target Line_204 (Cartesian target) at (-60.55, -1116.78, 243.45) mm, rotated rx 176.87 ry 0 rz -90 deg; joints [-1.125, 13.477, -25.633, 3.463, 114.965, -89.87] of Robot2
          - target Line_205 (Cartesian target) at (-60.55, -1114.25, 243.45) mm, rotated rx 176.87 ry 0 rz -90 deg; joints [-1.125, 13.477, -25.633, 3.463, 114.965, -89.87] of Robot2
          - target Line_206 (Cartesian target) at (-60.55, -1111.73, 243.45) mm, rotated rx 176.87 ry 0 rz -90 deg; joints [-1.125, 13.477, -25.633, 3.463, 114.965, -89.87] of Robot2
          - target Line_207 (Cartesian target) at (-60.55, -1109.2, 243.45) mm, rotated rx 176.87 ry 0 rz -90 deg; joints [-1.125, 13.477, -25.633, 3.463, 114.965, -89.87] of Robot2
          - target Line_208 (Cartesian target) at (-60.55, -1106.68, 243.45) mm, rotated rx 176.87 ry 0 rz -90 deg; joints [-1.125, 13.477, -25.633, 3.463, 114.965, -89.87] of Robot2
          - target Line_209 (Cartesian target) at (-60.55, -1104.15, 243.45) mm, rotated rx 176.87 ry 0 rz -90 deg; joints [-1.125, 13.477, -25.633, 3.463, 114.965, -89.87] of Robot2
          - target Line_210 (Cartesian target) at (-60.55, -1101.63, 243.45) mm, rotated rx 176.87 ry 0 rz -90 deg; joints [-1.125, 13.477, -25.633, 3.463, 114.965, -89.87] of Robot2
          - target Line_211 (Cartesian target) at (-60.55, -1099.1, 243.45) mm, rotated rx 176.87 ry 0 rz -90 deg; joints [-1.125, 13.477, -25.633, 3.463, 114.965, -89.87] of Robot2
          - target Line_212 (Cartesian target) at (-60.55, -1096.58, 243.45) mm, rotated rx 176.87 ry 0 rz -90 deg; joints [-1.125, 13.477, -25.633, 3.463, 114.965, -89.87] of Robot2
          - target Line_213 (Cartesian target) at (-60.55, -1094.05, 243.45) mm, rotated rx 176.87 ry 0 rz -90 deg; joints [-1.125, 13.477, -25.633, 3.463, 114.965, -89.87] of Robot2
          - target Line_214 (Cartesian target) at (-60.55, -1091.53, 243.45) mm, rotated rx 176.87 ry 0 rz -90 deg; joints [-1.125, 13.477, -25.633, 3.463, 114.965, -89.87] of Robot2
          - target Line_215 (Cartesian target) at (-60.55, -1089, 243.45) mm, rotated rx 176.87 ry 0 rz -90 deg; joints [-1.125, 13.477, -25.633, 3.463, 114.965, -89.87] of Robot2
          - target Line_216 (Cartesian target) at (-60.55, -1086.48, 243.45) mm, rotated rx 176.87 ry 0 rz -90 deg; joints [-1.125, 13.477, -25.633, 3.463, 114.965, -89.87] of Robot2
          - target Line_217 (Cartesian target) at (-60.55, -1083.95, 243.45) mm, rotated rx 176.87 ry 0 rz -90 deg; joints [-1.125, 13.477, -25.633, 3.463, 114.965, -89.87] of Robot2
          - target Line_218 (Cartesian target) at (-60.55, -1081.43, 243.45) mm, rotated rx 176.87 ry 0 rz -90 deg; joints [-1.125, 13.477, -25.633, 3.463, 114.965, -89.87] of Robot2
          - target Line_219 (Cartesian target) at (-60.55, -1078.9, 243.45) mm, rotated rx 176.87 ry 0 rz -90 deg; joints [-1.125, 13.477, -25.633, 3.463, 114.965, -89.87] of Robot2
          - target Line_220 (Cartesian target) at (-60.55, -1076.38, 243.45) mm, rotated rx 176.87 ry 0 rz -90 deg; joints [-1.125, 13.477, -25.633, 3.463, 114.965, -89.87] of Robot2
          - target Line_221 (Cartesian target) at (-60.55, -1073.85, 243.45) mm, rotated rx 176.87 ry 0 rz -90 deg; joints [-1.125, 13.477, -25.633, 3.463, 114.965, -89.87] of Robot2
          - target Line_222 (Cartesian target) at (-60.55, -1071.32, 243.45) mm, rotated rx 176.87 ry 0 rz -90 deg; joints [-1.125, 13.477, -25.633, 3.463, 114.965, -89.87] of Robot2
          - target Line_223 (Cartesian target) at (-60.55, -1068.8, 243.45) mm, rotated rx 176.87 ry 0 rz -90 deg; joints [-1.125, 13.477, -25.633, 3.463, 114.965, -89.87] of Robot2
          - target Line_224 (Cartesian target) at (-60.55, -1066.27, 243.45) mm, rotated rx 176.87 ry 0 rz -90 deg; joints [-1.125, 13.477, -25.633, 3.463, 114.965, -89.87] of Robot2
          - target Line_225 (Cartesian target) at (-60.55, -1063.75, 243.45) mm, rotated rx 176.87 ry 0 rz -90 deg; joints [-1.125, 13.477, -25.633, 3.463, 114.965, -89.87] of Robot2
          - target Line_226 (Cartesian target) at (-60.55, -1061.22, 243.45) mm, rotated rx 176.87 ry 0 rz -90 deg; joints [-1.125, 13.477, -25.633, 3.463, 114.965, -89.87] of Robot2
          - target Line_227 (Cartesian target) at (-60.55, -1058.7, 243.45) mm, rotated rx 176.87 ry 0 rz -90 deg; joints [-1.125, 13.477, -25.633, 3.463, 114.965, -89.87] of Robot2
          - target Line_228 (Cartesian target) at (-60.55, -1056.17, 243.45) mm, rotated rx 176.87 ry 0 rz -90 deg; joints [-1.125, 13.477, -25.633, 3.463, 114.965, -89.87] of Robot2
          - target Line_229 (Cartesian target) at (-60.55, -1053.65, 243.45) mm, rotated rx 176.87 ry 0 rz -90 deg; joints [-1.125, 13.477, -25.633, 3.463, 114.965, -89.87] of Robot2
          - target Line_230 (Cartesian target) at (-60.55, -1051.12, 243.45) mm, rotated rx 176.87 ry 0 rz -90 deg; joints [-1.125, 13.477, -25.633, 3.463, 114.965, -89.87] of Robot2
          - target Line_231 (Cartesian target) at (-60.55, -1048.6, 243.45) mm, rotated rx 176.87 ry 0 rz -90 deg; joints [-1.125, 13.477, -25.633, 3.463, 114.965, -89.87] of Robot2
          - target Line_232 (Cartesian target) at (-60.55, -1046.07, 243.45) mm, rotated rx 176.87 ry 0 rz -90 deg; joints [-1.125, 13.477, -25.633, 3.463, 114.965, -89.87] of Robot2
          - target Line_233 (Cartesian target) at (-60.55, -1043.55, 243.45) mm, rotated rx 176.87 ry 0 rz -90 deg; joints [-1.125, 13.477, -25.633, 3.463, 114.965, -89.87] of Robot2
          - target Line_234 (Cartesian target) at (-60.55, -1041.02, 243.45) mm, rotated rx 176.87 ry 0 rz -90 deg; joints [-1.125, 13.477, -25.633, 3.463, 114.965, -89.87] of Robot2
          - target Line_235 (Cartesian target) at (-60.55, -1038.5, 243.45) mm, rotated rx 176.87 ry 0 rz -90 deg; joints [-1.125, 13.477, -25.633, 3.463, 114.965, -89.87] of Robot2
          - target Line_236 (Cartesian target) at (-60.55, -1035.97, 243.45) mm, rotated rx 176.87 ry 0 rz -90 deg; joints [-1.125, 13.477, -25.633, 3.463, 114.965, -89.87] of Robot2
          - target Line_237 (Cartesian target) at (-60.55, -1033.45, 243.45) mm, rotated rx 176.87 ry 0 rz -90 deg; joints [-1.125, 13.477, -25.633, 3.463, 114.965, -89.87] of Robot2
          - target Line_238 (Cartesian target) at (-60.55, -1030.92, 243.45) mm, rotated rx 176.87 ry 0 rz -90 deg; joints [-1.125, 13.477, -25.633, 3.463, 114.965, -89.87] of Robot2
          - target Line_239 (Cartesian target) at (-60.55, -1028.4, 243.45) mm, rotated rx 176.87 ry 0 rz -90 deg; joints [-1.125, 13.477, -25.633, 3.463, 114.965, -89.87] of Robot2
          - target Line_240 (Cartesian target) at (-60.55, -1025.87, 243.45) mm, rotated rx 176.87 ry 0 rz -90 deg; joints [-1.125, 13.477, -25.633, 3.463, 114.965, -89.87] of Robot2
          - target Line_241 (Cartesian target) at (-60.55, -1023.34, 243.45) mm, rotated rx 176.87 ry 0 rz -90 deg; joints [-1.125, 13.477, -25.633, 3.463, 114.965, -89.87] of Robot2
          - target Line_242 (Cartesian target) at (-60.55, -1020.82, 243.45) mm, rotated rx 176.87 ry 0 rz -90 deg; joints [-1.125, 13.477, -25.633, 3.463, 114.965, -89.87] of Robot2
          - target Line_243 (Cartesian target) at (-60.55, -1018.29, 243.45) mm, rotated rx 176.87 ry 0 rz -90 deg; joints [-1.125, 13.477, -25.633, 3.463, 114.965, -89.87] of Robot2
          - target Line_244 (Cartesian target) at (-60.55, -1015.77, 243.45) mm, rotated rx 176.87 ry 0 rz -90 deg; joints [-1.125, 13.477, -25.633, 3.463, 114.965, -89.87] of Robot2
          - target Line_245 (Cartesian target) at (-60.55, -1013.24, 243.45) mm, rotated rx 176.87 ry 0 rz -90 deg; joints [-1.125, 13.477, -25.633, 3.463, 114.965, -89.87] of Robot2
          - target Line_246 (Cartesian target) at (-60.55, -1010.72, 243.45) mm, rotated rx 176.87 ry 0 rz -90 deg; joints [-1.125, 13.477, -25.633, 3.463, 114.965, -89.87] of Robot2
          - target Line_247 (Cartesian target) at (-60.55, -1008.19, 243.45) mm, rotated rx 176.87 ry 0 rz -90 deg; joints [-1.125, 13.477, -25.633, 3.463, 114.965, -89.87] of Robot2
          - target Line_248 (Cartesian target) at (-60.55, -1005.67, 243.45) mm, rotated rx 176.87 ry 0 rz -90 deg; joints [-1.125, 13.477, -25.633, 3.463, 114.965, -89.87] of Robot2
          - target Line_249 (Cartesian target) at (-60.55, -1003.14, 243.45) mm, rotated rx 176.87 ry 0 rz -90 deg; joints [-1.125, 13.477, -25.633, 3.463, 114.965, -89.87] of Robot2
          - target Line_250 (Cartesian target) at (-60.55, -1000.62, 243.45) mm, rotated rx 176.87 ry 0 rz -90 deg; joints [-1.125, 13.477, -25.633, 3.463, 114.965, -89.87] of Robot2
          - target Line_251 (Cartesian target) at (-60.55, -998.09, 243.45) mm, rotated rx 176.87 ry 0 rz -90 deg; joints [-1.125, 13.477, -25.633, 3.463, 114.965, -89.87] of Robot2
          - target Line_252 (Cartesian target) at (-60.55, -995.57, 243.45) mm, rotated rx 176.87 ry 0 rz -90 deg; joints [-1.125, 13.477, -25.633, 3.463, 114.965, -89.87] of Robot2
          - target Line_253 (Cartesian target) at (-60.55, -993.04, 243.45) mm, rotated rx 176.87 ry 0 rz -90 deg; joints [-1.125, 13.477, -25.633, 3.463, 114.965, -89.87] of Robot2
          - target Line_254 (Cartesian target) at (-60.55, -990.52, 243.45) mm, rotated rx 176.87 ry 0 rz -90 deg; joints [-1.125, 13.477, -25.633, 3.463, 114.965, -89.87] of Robot2
          - target Line_255 (Cartesian target) at (-60.55, -987.99, 243.45) mm, rotated rx 176.87 ry 0 rz -90 deg; joints [-1.125, 13.477, -25.633, 3.463, 114.965, -89.87] of Robot2
          - target Line_256 (Cartesian target) at (-60.55, -985.47, 243.45) mm, rotated rx 176.87 ry 0 rz -90 deg; joints [-1.125, 13.477, -25.633, 3.463, 114.965, -89.87] of Robot2
          - target Line_257 (Cartesian target) at (-60.55, -982.94, 243.45) mm, rotated rx 176.87 ry 0 rz -90 deg; joints [-1.125, 13.477, -25.633, 3.463, 114.965, -89.87] of Robot2
          - target Line_258 (Cartesian target) at (-60.55, -980.42, 243.45) mm, rotated rx 176.87 ry 0 rz -90 deg; joints [-1.125, 13.477, -25.633, 3.463, 114.965, -89.87] of Robot2
          - target Line_259 (Cartesian target) at (-60.55, -977.89, 243.45) mm, rotated rx 176.87 ry 0 rz -90 deg; joints [-1.125, 13.477, -25.633, 3.463, 114.965, -89.87] of Robot2
          - target Line_260 (Cartesian target) at (-60.55, -975.37, 243.45) mm, rotated rx 176.87 ry 0 rz -90 deg; joints [-1.125, 13.477, -25.633, 3.463, 114.965, -89.87] of Robot2
          - target Line_261 (Cartesian target) at (-60.55, -972.84, 243.45) mm, rotated rx 176.87 ry 0 rz -90 deg; joints [-1.125, 13.477, -25.633, 3.463, 114.965, -89.87] of Robot2
          - target Line_262 (Cartesian target) at (-60.55, -970.31, 243.45) mm, rotated rx 176.87 ry 0 rz -90 deg; joints [-1.125, 13.477, -25.633, 3.463, 114.965, -89.87] of Robot2
          - target Line_263 (Cartesian target) at (-60.55, -967.79, 243.45) mm, rotated rx 176.87 ry 0 rz -90 deg; joints [-1.125, 13.477, -25.633, 3.463, 114.965, -89.87] of Robot2
          - target Line_264 (Cartesian target) at (-60.55, -965.26, 243.45) mm, rotated rx 176.87 ry 0 rz -90 deg; joints [-1.125, 13.477, -25.633, 3.463, 114.965, -89.87] of Robot2
          - target Line_265 (Cartesian target) at (-60.55, -962.74, 243.45) mm, rotated rx 176.87 ry 0 rz -90 deg; joints [-1.125, 13.477, -25.633, 3.463, 114.965, -89.87] of Robot2
          - target Line_266 (Cartesian target) at (-60.55, -960.21, 243.45) mm, rotated rx 176.87 ry 0 rz -90 deg; joints [-1.125, 13.477, -25.633, 3.463, 114.965, -89.87] of Robot2
          - target Line_267 (Cartesian target) at (-60.55, -957.69, 243.45) mm, rotated rx 176.87 ry 0 rz -90 deg; joints [-1.125, 13.477, -25.633, 3.463, 114.965, -89.87] of Robot2
          - target Line_268 (Cartesian target) at (-60.55, -955.16, 243.45) mm, rotated rx 176.87 ry 0 rz -90 deg; joints [-1.125, 13.477, -25.633, 3.463, 114.965, -89.87] of Robot2
          - target Line_269 (Cartesian target) at (-60.55, -952.64, 243.45) mm, rotated rx 176.87 ry 0 rz -90 deg; joints [-1.125, 13.477, -25.633, 3.463, 114.965, -89.87] of Robot2
          - target Line_270 (Cartesian target) at (-60.55, -950.11, 243.45) mm, rotated rx 176.87 ry 0 rz -90 deg; joints [-1.125, 13.477, -25.633, 3.463, 114.965, -89.87] of Robot2
          - target Line_271 (Cartesian target) at (-60.55, -947.59, 243.45) mm, rotated rx 176.87 ry 0 rz -90 deg; joints [-1.125, 13.477, -25.633, 3.463, 114.965, -89.87] of Robot2
          - target Line_272 (Cartesian target) at (-60.55, -945.06, 243.45) mm, rotated rx 176.87 ry 0 rz -90 deg; joints [-1.125, 13.477, -25.633, 3.463, 114.965, -89.87] of Robot2
          - target Line_273 (Cartesian target) at (-60.55, -942.54, 243.45) mm, rotated rx 176.87 ry 0 rz -90 deg; joints [-1.125, 13.477, -25.633, 3.463, 114.965, -89.87] of Robot2
          - target Line_274 (Cartesian target) at (-60.55, -940.01, 243.45) mm, rotated rx 176.87 ry 0 rz -90 deg; joints [-1.125, 13.477, -25.633, 3.463, 114.965, -89.87] of Robot2
          - target Line_275 (Cartesian target) at (-60.55, -937.49, 243.45) mm, rotated rx 176.87 ry 0 rz -90 deg; joints [-1.125, 13.477, -25.633, 3.463, 114.965, -89.87] of Robot2
          - target Line_276 (Cartesian target) at (-60.55, -934.96, 243.45) mm, rotated rx 176.87 ry 0 rz -90 deg; joints [-1.125, 13.477, -25.633, 3.463, 114.965, -89.87] of Robot2
          - target Line_277 (Cartesian target) at (-60.55, -932.44, 243.45) mm, rotated rx 176.87 ry 0 rz -90 deg; joints [-1.125, 13.477, -25.633, 3.463, 114.965, -89.87] of Robot2
          - target Line_278 (Cartesian target) at (-60.55, -929.91, 243.45) mm, rotated rx 176.87 ry 0 rz -90 deg; joints [-1.125, 13.477, -25.633, 3.463, 114.965, -89.87] of Robot2
          - target Line_279 (Cartesian target) at (-60.55, -927.39, 243.45) mm, rotated rx 176.87 ry 0 rz -90 deg; joints [-1.125, 13.477, -25.633, 3.463, 114.965, -89.87] of Robot2
          - target Line_280 (Cartesian target) at (-60.55, -924.86, 243.45) mm, rotated rx 176.87 ry 0 rz -90 deg; joints [-1.125, 13.477, -25.633, 3.463, 114.965, -89.87] of Robot2
          - target Line_281 (Cartesian target) at (-60.55, -922.33, 243.45) mm, rotated rx 176.87 ry 0 rz -90 deg; joints [-1.125, 13.477, -25.633, 3.463, 114.965, -89.87] of Robot2
          - target Line_282 (Cartesian target) at (-60.55, -919.81, 243.45) mm, rotated rx 176.87 ry 0 rz -90 deg; joints [-1.125, 13.477, -25.633, 3.463, 114.965, -89.87] of Robot2
          - target Line_283 (Cartesian target) at (-60.55, -917.28, 243.45) mm, rotated rx 176.87 ry 0 rz -90 deg; joints [-1.125, 13.477, -25.633, 3.463, 114.965, -89.87] of Robot2
          - target Line_284 (Cartesian target) at (-60.55, -914.76, 243.45) mm, rotated rx 176.87 ry 0 rz -90 deg; joints [-1.125, 13.477, -25.633, 3.463, 114.965, -89.87] of Robot2
          - target Line_285 (Cartesian target) at (-60.55, -912.23, 243.45) mm, rotated rx 176.87 ry 0 rz -90 deg; joints [-1.125, 13.477, -25.633, 3.463, 114.965, -89.87] of Robot2
          - target Line_286 (Cartesian target) at (-60.55, -909.71, 243.45) mm, rotated rx 176.87 ry 0 rz -90 deg; joints [-1.125, 13.477, -25.633, 3.463, 114.965, -89.87] of Robot2
          - target Line_287 (Cartesian target) at (-60.55, -907.18, 243.45) mm, rotated rx 176.87 ry 0 rz -90 deg; joints [-1.125, 13.477, -25.633, 3.463, 114.965, -89.87] of Robot2
          - target Line_288 (Cartesian target) at (-60.55, -904.66, 243.45) mm, rotated rx 176.87 ry 0 rz -90 deg; joints [-1.125, 13.477, -25.633, 3.463, 114.965, -89.87] of Robot2
          - target Line_289 (Cartesian target) at (-60.55, -902.13, 243.45) mm, rotated rx 176.87 ry 0 rz -90 deg; joints [-1.125, 13.477, -25.633, 3.463, 114.965, -89.87] of Robot2
          - target Line_290 (Cartesian target) at (-60.55, -899.61, 243.45) mm, rotated rx 176.87 ry 0 rz -90 deg; joints [-1.125, 13.477, -25.633, 3.463, 114.965, -89.87] of Robot2
          - target Line_291 (Cartesian target) at (-60.55, -897.08, 243.45) mm, rotated rx 176.87 ry 0 rz -90 deg; joints [-1.125, 13.477, -25.633, 3.463, 114.965, -89.87] of Robot2
          - target Line_292 (Cartesian target) at (-60.55, -894.56, 243.45) mm, rotated rx 176.87 ry 0 rz -90 deg; joints [-1.125, 13.477, -25.633, 3.463, 114.965, -89.87] of Robot2
          - target Line_293 (Cartesian target) at (-60.55, -892.03, 243.45) mm, rotated rx 176.87 ry 0 rz -90 deg; joints [-1.125, 13.477, -25.633, 3.463, 114.965, -89.87] of Robot2
          - target Line_294 (Cartesian target) at (-60.55, -889.51, 243.45) mm, rotated rx 176.87 ry 0 rz -90 deg; joints [-1.125, 13.477, -25.633, 3.463, 114.965, -89.87] of Robot2
          - target Line_295 (Cartesian target) at (-60.55, -886.98, 243.45) mm, rotated rx 176.87 ry 0 rz -90 deg; joints [-1.125, 13.477, -25.633, 3.463, 114.965, -89.87] of Robot2
          - target Line_296 (Cartesian target) at (-60.55, -884.46, 243.45) mm, rotated rx 176.87 ry 0 rz -90 deg; joints [-1.125, 13.477, -25.633, 3.463, 114.965, -89.87] of Robot2
          - target Line_297 (Cartesian target) at (-60.55, -881.93, 243.45) mm, rotated rx 176.87 ry 0 rz -90 deg; joints [-1.125, 13.477, -25.633, 3.463, 114.965, -89.87] of Robot2
          - target Line_298 (Cartesian target) at (-60.55, -879.41, 243.45) mm, rotated rx 176.87 ry 0 rz -90 deg; joints [-1.125, 13.477, -25.633, 3.463, 114.965, -89.87] of Robot2
          - target Line_299 (Cartesian target) at (-60.55, -876.88, 243.45) mm, rotated rx 176.87 ry 0 rz -90 deg; joints [-1.125, 13.477, -25.633, 3.463, 114.965, -89.87] of Robot2
          - target Line_300 (Cartesian target) at (-60.55, -874.35, 243.45) mm, rotated rx 176.87 ry 0 rz -90 deg; joints [-1.125, 13.477, -25.633, 3.463, 114.965, -89.87] of Robot2
          - target Line_301 (Cartesian target) at (-60.55, -874.35, 243.45) mm, rotated rx 176.87 ry 0.69 rz -90.24 deg; joints [-1.125, 13.477, -25.633, 3.463, 114.965, -89.87] of Robot2
          - target Line_302 (Cartesian target) at (-59.3, -874.35, 243.45) mm, rotated rx 176.87 ry 0.69 rz -90.24 deg; joints [-1.125, 13.477, -25.633, 3.463, 114.965, -89.87] of Robot2
          - target Line_303 (Cartesian target) at (-58.05, -874.35, 243.45) mm, rotated rx 176.87 ry 0.69 rz -90.24 deg; joints [-1.125, 13.477, -25.633, 3.463, 114.965, -89.87] of Robot2
          - target Line_304 (Cartesian target) at (-56.79, -874.35, 243.45) mm, rotated rx 176.87 ry 0.69 rz -90.24 deg; joints [-1.125, 13.477, -25.633, 3.463, 114.965, -89.87] of Robot2
          - target Line_305 (Cartesian target) at (-55.54, -874.35, 243.45) mm, rotated rx 176.87 ry 0.69 rz -90.24 deg; joints [-1.125, 13.477, -25.633, 3.463, 114.965, -89.87] of Robot2
          - target Line_306 (Cartesian target) at (-54.29, -874.35, 243.45) mm, rotated rx 176.87 ry 0.69 rz -90.24 deg; joints [-1.125, 13.477, -25.633, 3.463, 114.965, -89.87] of Robot2
          - target Line_307 (Cartesian target) at (-53.04, -874.35, 243.45) mm, rotated rx 176.87 ry 0.69 rz -90.24 deg; joints [-1.125, 13.477, -25.633, 3.463, 114.965, -89.87] of Robot2
          - target Line_308 (Cartesian target) at (-51.78, -874.35, 243.45) mm, rotated rx 176.87 ry 0.69 rz -90.24 deg; joints [-1.125, 13.477, -25.633, 3.463, 114.965, -89.87] of Robot2
          - target Line_309 (Cartesian target) at (-50.53, -874.35, 243.45) mm, rotated rx 176.87 ry 0.69 rz -90.24 deg; joints [-1.125, 13.477, -25.633, 3.463, 114.965, -89.87] of Robot2
          - target Line_310 (Cartesian target) at (-49.28, -874.35, 243.45) mm, rotated rx 176.87 ry 0.69 rz -90.24 deg; joints [-1.125, 13.477, -25.633, 3.463, 114.965, -89.87] of Robot2
          - target Line_311 (Cartesian target) at (-48.03, -874.35, 243.45) mm, rotated rx 176.87 ry 0.69 rz -90.24 deg; joints [-1.125, 13.477, -25.633, 3.463, 114.965, -89.87] of Robot2
          - target Line_312 (Cartesian target) at (-46.77, -874.35, 243.45) mm, rotated rx 176.87 ry 0.69 rz -90.24 deg; joints [-1.125, 13.477, -25.633, 3.463, 114.965, -89.87] of Robot2
          - target Line_313 (Cartesian target) at (-45.52, -874.35, 243.45) mm, rotated rx 176.87 ry 0.69 rz -90.24 deg; joints [-1.125, 13.477, -25.633, 3.463, 114.965, -89.87] of Robot2
          - target Line_314 (Cartesian target) at (-44.27, -874.35, 243.45) mm, rotated rx 176.87 ry 0.69 rz -90.24 deg; joints [-1.125, 13.477, -25.633, 3.463, 114.965, -89.87] of Robot2
          - target Line_315 (Cartesian target) at (-43.02, -874.35, 243.45) mm, rotated rx 176.87 ry 0.69 rz -90.24 deg; joints [-1.125, 13.477, -25.633, 3.463, 114.965, -89.87] of Robot2
          - target Line_316 (Cartesian target) at (-41.76, -874.35, 243.45) mm, rotated rx 176.87 ry 0.69 rz -90.24 deg; joints [-1.125, 13.477, -25.633, 3.463, 114.965, -89.87] of Robot2
          - target Line_317 (Cartesian target) at (-40.51, -874.35, 243.45) mm, rotated rx 176.87 ry 0.69 rz -90.24 deg; joints [-1.125, 13.477, -25.633, 3.463, 114.965, -89.87] of Robot2
          - target Line_318 (Cartesian target) at (-39.26, -874.35, 243.45) mm, rotated rx 176.87 ry 0.69 rz -90.24 deg; joints [-1.125, 13.477, -25.633, 3.463, 114.965, -89.87] of Robot2
          - target Line_319 (Cartesian target) at (-38.01, -874.35, 243.45) mm, rotated rx 176.87 ry 0.69 rz -90.24 deg; joints [-1.125, 13.477, -25.633, 3.463, 114.965, -89.87] of Robot2
          - target Line_320 (Cartesian target) at (-36.75, -874.35, 243.45) mm, rotated rx 176.87 ry 0.69 rz -90.24 deg; joints [-1.125, 13.477, -25.633, 3.463, 114.965, -89.87] of Robot2
          - target Line_321 (Cartesian target) at (-35.5, -874.35, 243.45) mm, rotated rx 176.87 ry 0.69 rz -90.24 deg; joints [-1.125, 13.477, -25.633, 3.463, 114.965, -89.87] of Robot2
          - target Line_322 (Cartesian target) at (-34.25, -874.35, 243.45) mm, rotated rx 176.87 ry 0.69 rz -90.24 deg; joints [-1.125, 13.477, -25.633, 3.463, 114.965, -89.87] of Robot2
          - target Line_323 (Cartesian target) at (-33, -874.35, 243.45) mm, rotated rx 176.87 ry 0.69 rz -90.24 deg; joints [-1.125, 13.477, -25.633, 3.463, 114.965, -89.87] of Robot2
          - target Line_324 (Cartesian target) at (-31.74, -874.35, 243.45) mm, rotated rx 176.87 ry 0.69 rz -90.24 deg; joints [-1.125, 13.477, -25.633, 3.463, 114.965, -89.87] of Robot2
          - target Line_325 (Cartesian target) at (-30.49, -874.35, 243.45) mm, rotated rx 176.87 ry 0.69 rz -90.24 deg; joints [-1.125, 13.477, -25.633, 3.463, 114.965, -89.87] of Robot2
          - target Line_326 (Cartesian target) at (-29.24, -874.35, 243.45) mm, rotated rx 176.87 ry 0.69 rz -90.24 deg; joints [-1.125, 13.477, -25.633, 3.463, 114.965, -89.87] of Robot2
          - target Line_327 (Cartesian target) at (-27.99, -874.35, 243.45) mm, rotated rx 176.87 ry 0.69 rz -90.24 deg; joints [-1.125, 13.477, -25.633, 3.463, 114.965, -89.87] of Robot2
          - target Line_328 (Cartesian target) at (-26.73, -874.35, 243.45) mm, rotated rx 176.87 ry 0.69 rz -90.24 deg; joints [-1.125, 13.477, -25.633, 3.463, 114.965, -89.87] of Robot2
          - target Line_329 (Cartesian target) at (-25.48, -874.35, 243.45) mm, rotated rx 176.87 ry 0.69 rz -90.24 deg; joints [-1.125, 13.477, -25.633, 3.463, 114.965, -89.87] of Robot2
          - target Line_330 (Cartesian target) at (-24.23, -874.35, 243.45) mm, rotated rx 176.87 ry 0.69 rz -90.24 deg; joints [-1.125, 13.477, -25.633, 3.463, 114.965, -89.87] of Robot2
          - target Line_331 (Cartesian target) at (-22.98, -874.35, 243.45) mm, rotated rx 176.87 ry 0.69 rz -90.24 deg; joints [-1.125, 13.477, -25.633, 3.463, 114.965, -89.87] of Robot2
          - target Line_332 (Cartesian target) at (-21.72, -874.35, 243.45) mm, rotated rx 176.87 ry 0.69 rz -90.24 deg; joints [-1.125, 13.477, -25.633, 3.463, 114.965, -89.87] of Robot2
          - target Line_333 (Cartesian target) at (-20.47, -874.35, 243.45) mm, rotated rx 176.87 ry 0.69 rz -90.24 deg; joints [-1.125, 13.477, -25.633, 3.463, 114.965, -89.87] of Robot2
          - target Line_334 (Cartesian target) at (-19.22, -874.35, 243.45) mm, rotated rx 176.87 ry 0.69 rz -90.24 deg; joints [-1.125, 13.477, -25.633, 3.463, 114.965, -89.87] of Robot2
          - target Line_335 (Cartesian target) at (-17.97, -874.35, 243.45) mm, rotated rx 176.87 ry 0.69 rz -90.24 deg; joints [-1.125, 13.477, -25.633, 3.463, 114.965, -89.87] of Robot2
          - target Line_336 (Cartesian target) at (-16.71, -874.35, 243.45) mm, rotated rx 176.87 ry 0.69 rz -90.24 deg; joints [-1.125, 13.477, -25.633, 3.463, 114.965, -89.87] of Robot2
          - target Line_337 (Cartesian target) at (-15.46, -874.35, 243.45) mm, rotated rx 176.87 ry 0.69 rz -90.24 deg; joints [-1.125, 13.477, -25.633, 3.463, 114.965, -89.87] of Robot2
          - target Line_338 (Cartesian target) at (-14.21, -874.35, 243.45) mm, rotated rx 176.87 ry 0.69 rz -90.24 deg; joints [-1.125, 13.477, -25.633, 3.463, 114.965, -89.87] of Robot2
          - target Line_339 (Cartesian target) at (-12.96, -874.35, 243.45) mm, rotated rx 176.87 ry 0.69 rz -90.24 deg; joints [-1.125, 13.477, -25.633, 3.463, 114.965, -89.87] of Robot2
          - target Line_340 (Cartesian target) at (-11.7, -874.35, 243.45) mm, rotated rx 176.87 ry 0.69 rz -90.24 deg; joints [-1.125, 13.477, -25.633, 3.463, 114.965, -89.87] of Robot2
          - target Line_341 (Cartesian target) at (-10.45, -874.35, 243.45) mm, rotated rx 176.87 ry 0.69 rz -90.24 deg; joints [-1.125, 13.477, -25.633, 3.463, 114.965, -89.87] of Robot2
          - target Line_342 (Cartesian target) at (-9.2, -874.35, 243.45) mm, rotated rx 176.87 ry 0.69 rz -90.24 deg; joints [-1.125, 13.477, -25.633, 3.463, 114.965, -89.87] of Robot2
          - target Line_343 (Cartesian target) at (-7.95, -874.35, 243.45) mm, rotated rx 176.87 ry 0.69 rz -90.24 deg; joints [-1.125, 13.477, -25.633, 3.463, 114.965, -89.87] of Robot2
          - target Line_344 (Cartesian target) at (-6.69, -874.35, 243.45) mm, rotated rx 176.87 ry 0.69 rz -90.24 deg; joints [-1.125, 13.477, -25.633, 3.463, 114.965, -89.87] of Robot2
          - target Line_345 (Cartesian target) at (-5.44, -874.35, 243.45) mm, rotated rx 176.87 ry 0.69 rz -90.24 deg; joints [-1.125, 13.477, -25.633, 3.463, 114.965, -89.87] of Robot2
          - target Line_346 (Cartesian target) at (-4.19, -874.35, 243.45) mm, rotated rx 176.87 ry 0.69 rz -90.24 deg; joints [-1.125, 13.477, -25.633, 3.463, 114.965, -89.87] of Robot2
          - target Line_347 (Cartesian target) at (-2.94, -874.35, 243.45) mm, rotated rx 176.87 ry 0.69 rz -90.24 deg; joints [-1.125, 13.477, -25.633, 3.463, 114.965, -89.87] of Robot2
          - target Line_348 (Cartesian target) at (-1.68, -874.35, 243.45) mm, rotated rx 176.87 ry 0.69 rz -90.24 deg; joints [-1.125, 13.477, -25.633, 3.463, 114.965, -89.87] of Robot2
          - target Line_349 (Cartesian target) at (-0.43, -874.35, 243.45) mm, rotated rx 176.87 ry 0.69 rz -90.24 deg; joints [-1.125, 13.477, -25.633, 3.463, 114.965, -89.87] of Robot2
          - target Line_350 (Cartesian target) at (0.82, -874.35, 243.45) mm, rotated rx 176.87 ry 0.69 rz -90.24 deg; joints [-1.125, 13.477, -25.633, 3.463, 114.965, -89.87] of Robot2
          - target Line_351 (Cartesian target) at (2.07, -874.35, 243.45) mm, rotated rx 176.87 ry 0.69 rz -90.24 deg; joints [-1.125, 13.477, -25.633, 3.463, 114.965, -89.87] of Robot2
          - target Line_352 (Cartesian target) at (3.33, -874.35, 243.45) mm, rotated rx 176.87 ry 0.69 rz -90.24 deg; joints [-1.125, 13.477, -25.633, 3.463, 114.965, -89.87] of Robot2
          - target Line_353 (Cartesian target) at (4.58, -874.35, 243.45) mm, rotated rx 176.87 ry 0.69 rz -90.24 deg; joints [-1.125, 13.477, -25.633, 3.463, 114.965, -89.87] of Robot2
          - target Line_354 (Cartesian target) at (5.83, -874.35, 243.45) mm, rotated rx 176.87 ry 0.69 rz -90.24 deg; joints [-1.125, 13.477, -25.633, 3.463, 114.965, -89.87] of Robot2
          - target Line_355 (Cartesian target) at (7.08, -874.35, 243.45) mm, rotated rx 176.87 ry 0.69 rz -90.24 deg; joints [-1.125, 13.477, -25.633, 3.463, 114.965, -89.87] of Robot2
          - target Line_356 (Cartesian target) at (8.34, -874.35, 243.45) mm, rotated rx 176.87 ry 0.69 rz -90.24 deg; joints [-1.125, 13.477, -25.633, 3.463, 114.965, -89.87] of Robot2
          - target Line_357 (Cartesian target) at (9.59, -874.35, 243.45) mm, rotated rx 176.87 ry 0.69 rz -90.24 deg; joints [-1.125, 13.477, -25.633, 3.463, 114.965, -89.87] of Robot2
          - target Line_358 (Cartesian target) at (10.84, -874.35, 243.45) mm, rotated rx 176.87 ry 0.69 rz -90.24 deg; joints [-1.125, 13.477, -25.633, 3.463, 114.965, -89.87] of Robot2
          - target Line_359 (Cartesian target) at (12.09, -874.35, 243.45) mm, rotated rx 176.87 ry 0.69 rz -90.24 deg; joints [-1.125, 13.477, -25.633, 3.463, 114.965, -89.87] of Robot2
          - target Line_360 (Cartesian target) at (13.35, -874.35, 243.45) mm, rotated rx 176.87 ry 0.69 rz -90.24 deg; joints [-1.125, 13.477, -25.633, 3.463, 114.965, -89.87] of Robot2
          - target Line_361 (Cartesian target) at (14.6, -874.35, 243.45) mm, rotated rx 176.87 ry 0.69 rz -90.24 deg; joints [-1.125, 13.477, -25.633, 3.463, 114.965, -89.87] of Robot2
          - target Line_362 (Cartesian target) at (15.85, -874.35, 243.45) mm, rotated rx 176.87 ry 0.69 rz -90.24 deg; joints [-1.125, 13.477, -25.633, 3.463, 114.965, -89.87] of Robot2
          - target Line_363 (Cartesian target) at (17.1, -874.35, 243.45) mm, rotated rx 176.87 ry 0.69 rz -90.24 deg; joints [-1.125, 13.477, -25.633, 3.463, 114.965, -89.87] of Robot2
          - target Line_364 (Cartesian target) at (18.36, -874.35, 243.45) mm, rotated rx 176.87 ry 0.69 rz -90.24 deg; joints [-1.125, 13.477, -25.633, 3.463, 114.965, -89.87] of Robot2
          - target Line_365 (Cartesian target) at (19.61, -874.35, 243.45) mm, rotated rx 176.87 ry 0.69 rz -90.24 deg; joints [-1.125, 13.477, -25.633, 3.463, 114.965, -89.87] of Robot2
          - target Line_366 (Cartesian target) at (20.86, -874.35, 243.45) mm, rotated rx 176.87 ry 0.69 rz -90.24 deg; joints [-1.125, 13.477, -25.633, 3.463, 114.965, -89.87] of Robot2
          - target Line_367 (Cartesian target) at (22.11, -874.35, 243.45) mm, rotated rx 176.87 ry 0.69 rz -90.24 deg; joints [-1.125, 13.477, -25.633, 3.463, 114.965, -89.87] of Robot2
          - target Line_368 (Cartesian target) at (23.37, -874.35, 243.45) mm, rotated rx 176.87 ry 0.69 rz -90.24 deg; joints [-1.125, 13.477, -25.633, 3.463, 114.965, -89.87] of Robot2
          - target Line_369 (Cartesian target) at (24.62, -874.35, 243.45) mm, rotated rx 176.87 ry 0.69 rz -90.24 deg; joints [-1.125, 13.477, -25.633, 3.463, 114.965, -89.87] of Robot2
          - target Line_370 (Cartesian target) at (25.87, -874.35, 243.45) mm, rotated rx 176.87 ry 0.69 rz -90.24 deg; joints [-1.125, 13.477, -25.633, 3.463, 114.965, -89.87] of Robot2
          - target Line_371 (Cartesian target) at (27.12, -874.35, 243.45) mm, rotated rx 176.87 ry 0.69 rz -90.24 deg; joints [-1.125, 13.477, -25.633, 3.463, 114.965, -89.87] of Robot2
          - target Line_372 (Cartesian target) at (28.38, -874.35, 243.45) mm, rotated rx 176.87 ry 0.69 rz -90.24 deg; joints [-1.125, 13.477, -25.633, 3.463, 114.965, -89.87] of Robot2
          - target Line_373 (Cartesian target) at (29.63, -874.35, 243.45) mm, rotated rx 176.87 ry 0.69 rz -90.24 deg; joints [-1.125, 13.477, -25.633, 3.463, 114.965, -89.87] of Robot2
          - target Line_374 (Cartesian target) at (30.88, -874.35, 243.45) mm, rotated rx 176.87 ry 0.69 rz -90.24 deg; joints [-1.125, 13.477, -25.633, 3.463, 114.965, -89.87] of Robot2
          - target Line_375 (Cartesian target) at (32.13, -874.35, 243.45) mm, rotated rx 176.87 ry 0.69 rz -90.24 deg; joints [-1.125, 13.477, -25.633, 3.463, 114.965, -89.87] of Robot2
          - target Line_376 (Cartesian target) at (33.39, -874.35, 243.45) mm, rotated rx 176.87 ry 0.69 rz -90.24 deg; joints [-1.125, 13.477, -25.633, 3.463, 114.965, -89.87] of Robot2
          - target Line_377 (Cartesian target) at (34.64, -874.35, 243.45) mm, rotated rx 176.87 ry 0.69 rz -90.24 deg; joints [-1.125, 13.477, -25.633, 3.463, 114.965, -89.87] of Robot2
          - target Line_378 (Cartesian target) at (35.89, -874.35, 243.45) mm, rotated rx 176.87 ry 0.69 rz -90.24 deg; joints [-1.125, 13.477, -25.633, 3.463, 114.965, -89.87] of Robot2
          - target Line_379 (Cartesian target) at (37.14, -874.35, 243.45) mm, rotated rx 176.87 ry 0.69 rz -90.24 deg; joints [-1.125, 13.477, -25.633, 3.463, 114.965, -89.87] of Robot2
          - target Line_380 (Cartesian target) at (38.4, -874.35, 243.45) mm, rotated rx 176.87 ry 0.69 rz -90.24 deg; joints [-1.125, 13.477, -25.633, 3.463, 114.965, -89.87] of Robot2
          - target Line_381 (Cartesian target) at (39.65, -874.35, 243.45) mm, rotated rx 176.87 ry 0.69 rz -90.24 deg; joints [-1.125, 13.477, -25.633, 3.463, 114.965, -89.87] of Robot2
          - target Line_382 (Cartesian target) at (40.9, -874.35, 243.45) mm, rotated rx 176.87 ry 0.69 rz -90.24 deg; joints [-1.125, 13.477, -25.633, 3.463, 114.965, -89.87] of Robot2
          - target Line_383 (Cartesian target) at (42.16, -874.35, 243.45) mm, rotated rx 176.87 ry 0.69 rz -90.24 deg; joints [-1.125, 13.477, -25.633, 3.463, 114.965, -89.87] of Robot2
          - target Line_384 (Cartesian target) at (43.41, -874.35, 243.45) mm, rotated rx 176.87 ry 0.69 rz -90.24 deg; joints [-1.125, 13.477, -25.633, 3.463, 114.965, -89.87] of Robot2
          - target Line_385 (Cartesian target) at (44.66, -874.35, 243.45) mm, rotated rx 176.87 ry 0.69 rz -90.24 deg; joints [-1.125, 13.477, -25.633, 3.463, 114.965, -89.87] of Robot2
          - target Line_386 (Cartesian target) at (45.91, -874.35, 243.45) mm, rotated rx 176.87 ry 0.69 rz -90.24 deg; joints [-1.125, 13.477, -25.633, 3.463, 114.965, -89.87] of Robot2
          - target Line_387 (Cartesian target) at (47.17, -874.35, 243.45) mm, rotated rx 176.87 ry 0.69 rz -90.24 deg; joints [-1.125, 13.477, -25.633, 3.463, 114.965, -89.87] of Robot2
          - target Line_388 (Cartesian target) at (48.42, -874.35, 243.45) mm, rotated rx 176.87 ry 0.69 rz -90.24 deg; joints [-1.125, 13.477, -25.633, 3.463, 114.965, -89.87] of Robot2
          - target Line_389 (Cartesian target) at (49.67, -874.35, 243.45) mm, rotated rx 176.87 ry 0.69 rz -90.24 deg; joints [-1.125, 13.477, -25.633, 3.463, 114.965, -89.87] of Robot2
          - target Line_390 (Cartesian target) at (50.92, -874.35, 243.45) mm, rotated rx 176.87 ry 0.69 rz -90.24 deg; joints [-1.125, 13.477, -25.633, 3.463, 114.965, -89.87] of Robot2
          - target Line_391 (Cartesian target) at (52.18, -874.35, 243.45) mm, rotated rx 176.87 ry 0.69 rz -90.24 deg; joints [-1.125, 13.477, -25.633, 3.463, 114.965, -89.87] of Robot2
          - target Line_392 (Cartesian target) at (53.43, -874.35, 243.45) mm, rotated rx 176.87 ry 0.69 rz -90.24 deg; joints [-1.125, 13.477, -25.633, 3.463, 114.965, -89.87] of Robot2
          - target Line_393 (Cartesian target) at (54.68, -874.35, 243.45) mm, rotated rx 176.87 ry 0.69 rz -90.24 deg; joints [-1.125, 13.477, -25.633, 3.463, 114.965, -89.87] of Robot2
          - target Line_394 (Cartesian target) at (55.93, -874.35, 243.45) mm, rotated rx 176.87 ry 0.69 rz -90.24 deg; joints [-1.125, 13.477, -25.633, 3.463, 114.965, -89.87] of Robot2
          - target Line_395 (Cartesian target) at (57.19, -874.35, 243.45) mm, rotated rx 176.87 ry 0.69 rz -90.24 deg; joints [-1.125, 13.477, -25.633, 3.463, 114.965, -89.87] of Robot2
          - target Line_396 (Cartesian target) at (58.44, -874.35, 243.45) mm, rotated rx 176.87 ry 0.69 rz -90.24 deg; joints [-1.125, 13.477, -25.633, 3.463, 114.965, -89.87] of Robot2
          - target Line_397 (Cartesian target) at (59.69, -874.35, 243.45) mm, rotated rx 176.87 ry 0.69 rz -90.24 deg; joints [-1.125, 13.477, -25.633, 3.463, 114.965, -89.87] of Robot2
          - target Line_398 (Cartesian target) at (60.94, -874.35, 243.45) mm, rotated rx 176.87 ry 0.69 rz -90.24 deg; joints [-1.125, 13.477, -25.633, 3.463, 114.965, -89.87] of Robot2
          - target Line_399 (Cartesian target) at (62.2, -874.35, 243.45) mm, rotated rx 176.87 ry 0.69 rz -90.24 deg; joints [-1.125, 13.477, -25.633, 3.463, 114.965, -89.87] of Robot2
          - target Line_400 (Cartesian target) at (63.45, -874.35, 243.45) mm, rotated rx 176.87 ry 0.69 rz -90.24 deg; joints [-1.125, 13.477, -25.633, 3.463, 114.965, -89.87] of Robot2
        - tool OnRobot VGC10 Vacuum Gripper, TCP at (0, 0, 117.4) mm, size 100 x 100 x 114.9 mm
          - object Kocka_Frame at (0, 0, 0) mm, size 125 x 250 x 125 mm, geometry from Prism-250x125x125mm.sld
      - target Start_Robot1 (Cartesian target) at (572.58, -0.43, 476.33) mm, rotated rx -0.7 ry -3.12 rz -89.76 deg; joints [-1.125, 13.477, -25.633, 3.463, 114.965, -89.87] of Robot1
      - target Target 2 (Cartesian target) at (823.05, 20.7, 472.16) mm, rotated rx -0.7 ry -3.12 rz -89.76 deg; joints [0.694, 56.157, -3.158, 3.121, 92.427, -89.379] of Robot1
      - target Target 3 (Cartesian target) at (703.44, 0.04, 474.73) mm, rotated rx -0.7 ry -3.12 rz -89.76 deg; joints [-0.877, 32.302, -18.707, 3.299, 108.038, -90.062] of Robot1
      - target Target 4 (Cartesian target) at (823.73, -139.92, 480.93) mm, rotated rx -0.7 ry -3.12 rz -89.76 deg; joints [-10.396, 62.751, 3.614, 3.206, 86.279, -100.826] of Robot1
      - target Target 5 (Cartesian target) at (822.19, 221.97, 461.18) mm, rotated rx -0.7 ry -3.12 rz -89.76 deg; joints [14.446, 67.836, 5.39, 2.876, 83.171, -76.085] of Robot1
      - target Target 6 (Cartesian target) at (823.05, 20.7, 472.16) mm, rotated rx 3.13 ry -0.69 rz -179.94 deg; joints [0.694, 56.157, -3.158, 3.121, 92.427, 0.763] of Robot1
      - target Target 7 (Cartesian target) at (823.05, 20.7, 472.16) mm, rotated rx 3.26 ry -16.51 rz 179.17 deg; joints [0.768, 43.474, -11.338, 2.818, 84.754, 1.273] of Robot1
      - target Target 8 (Cartesian target) at (823.05, 20.7, 472.16) mm, rotated rx 3.14 ry 5.76 rz -179.58 deg; joints [0.682, 67.782, 7.057, 3.169, 88.695, 0.191] of Robot1
      - target Target 9 (Cartesian target) at (817.23, 11.21, 338.48) mm, rotated rx 3.13 ry -1.92 rz 180 deg; joints [0.031, 55.107, -22.461, 3.338, 110.511, 1.205] of Robot1
      - target Target 10 (Cartesian target) at (824.79, 23.54, 524.1) mm, rotated rx 3.13 ry -1.92 rz 180 deg; joints [0.894, 59.955, 7.349, 3.138, 80.698, 0.391] of Robot1
      - target Target 11 (Cartesian target) at (701.54, 23.55, 528.23) mm, rotated rx 3.13 ry -1.92 rz 180 deg; joints [1.054, 30.576, -12.175, 3.141, 100.185, 1.614] of Robot1
      - target Target 12 (Cartesian target) at (701.54, 23.55, 528.23) mm, rotated rx 3.72 ry -32.84 rz 178.08 deg; joints [1.38, 14.981, -13.624, 2.044, 70.66, 2.095] of Robot1
      - target TMP_R1 (Cartesian target) at (700, -56.46, 604.1) mm, rotated rx 180 ry -0.01 rz -179.76 deg; joints [6.118, 22.277, -53.703, 0.008, -36.284, -5.881] of Robot2
      - target TMP_R2 (Cartesian target) at (700, -56.46, 604.1) mm, rotated rx 180 ry -0.01 rz -179.76 deg; joints [6.118, 22.277, -53.703, 180.008, 36.284, 174.119] of Robot2
      - target TMP_R3 (Cartesian target) at (700, -56.46, 604.1) mm, rotated rx 180 ry -0.01 rz -179.76 deg; joints [6.118, 22.277, -53.703, 180.008, 36.284, -185.881] of Robot2
  - frame Pozicija 2 at (2320, 0, 840) mm
    - frame Robot2 at (0, 1000, 330) mm, rotated rx 0 ry 0 rz -180 deg
      - robot Robot2: 6 axes
          modified DH rows (alpha deg, a mm, theta deg, d mm): 0, 0, 0, 330; -90, 75, -90, 0; 0, 400, 0, 0; -90, 75, 0, 410; 90, 0, 0, 0; -90, 0, 0, 80
          base shift (0, 0, -330) mm
          joint limits [-170, -60, -70, -190, -115, -400] to [170, 140, 170, 190, 115, 400]; home [0, 0, 0, 0, 0, 0]; saved at [6.118, 22.277, -53.703, 0.008, -36.284, -5.881]
        - tool Robot2, TCP at (0, 0, 0) mm
  - Python program Target_Generator (listed below)
  - Python program Line_Following (listed below)
  - Python program Line_Following_konfg (listed below)
  - Python program Line_Following_Analiza (listed below)
  - Python program Line_Following_ReplayAnalize (listed below)
  - program Program_R1 (39 instructions, listed below)
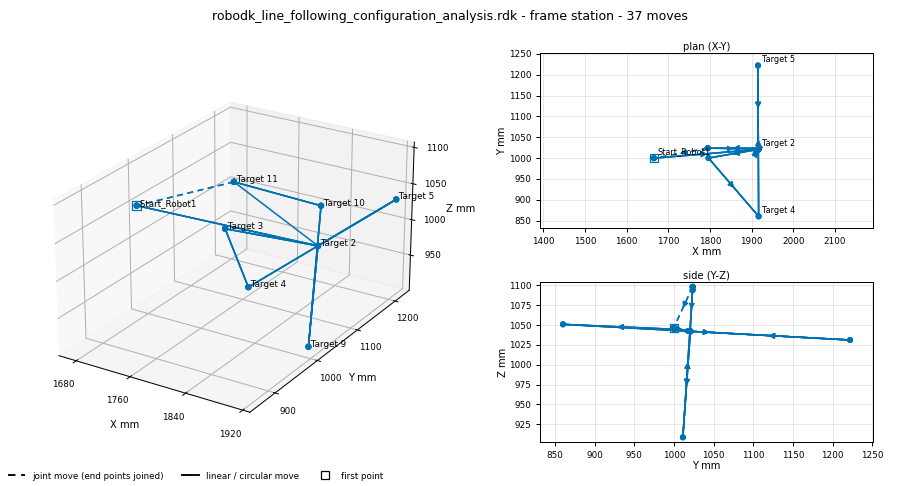
[picture p0: tool path of robodk_line_following_configuration_analysis.rdk in frame station, 37 of 37 moves have a stored position in this frame; points joined in program order, loops and branches not executed]

--- Python program Target_Generator ---
from robodk.robolink import *
from robodk.robomath import *

RDK = Robolink()

START_NAME = 'Kut_4'
END_NAME   = 'Pocetak'
PREFIX     = 'Line_'
NPTS       = 100

START_NUM  = 301    # <-- nova numeracija: 201-400
UPDATE_IF_EXISTS = True   # <-- ako postoji Line_2xx, samo ga update-a

tA = RDK.Item(START_NAME, ITEM_TYPE_TARGET)
tB = RDK.Item(END_NAME, ITEM_TYPE_TARGET)
if not tA.Valid(): raise Exception(f"Ne postoji target: {START_NAME}")
if not tB.Valid(): raise Exception(f"Ne postoji target: {END_NAME}")

parent = tA.Parent()
if not parent.Valid():
    raise Exception("Pocetak nema Parent() -> stavi Pocetak pod frame/predmet u tree-u")

TA = tA.Pose()
TB = tB.Pose()

xa, ya, za, rxa, rya, rza = pose_2_xyzrpw(TA)
xb, yb, zb, _,   _,   _   = pose_2_xyzrpw(TB)

dx, dy, dz = xb-xa, yb-ya, zb-za
print(f"Pocetak XYZ: {xa:.3f}, {ya:.3f}, {za:.3f}")
print(f"Kraj    XYZ: {xb:.3f}, {yb:.3f}, {zb:.3f}")
print(f"Delta XYZ:   {dx:.3f}, {dy:.3f}, {dz:.3f}")

adx, ady, adz = abs(dx), abs(dy), abs(dz)
if adx >= ady and adx >= adz:
    axis = 'X'; a0, a1 = xa, xb
elif ady >= adx and ady >= adz:
    axis = 'Y'; a0, a1 = ya, yb
else:
    axis = 'Z'; a0, a1 = za, zb
print(f"Interpoliram SAMO os {axis}: {a0:.3f} -> {a1:.3f}")

for i in range(NPTS):
    s = i/(NPTS-1) if NPTS > 1 else 0.0
    aval = a0 + (a1-a0)*s

    x, y, z = xa, ya, za
    if axis == 'X': x = aval
    if axis == 'Y': y = aval
    if axis == 'Z': z = aval

    Ti = xyzrpw_2_pose([x, y, z, rxa, rya, rza])

    num = START_NUM + i
    name = f"{PREFIX}{num:03d}"  # Line_201 ... Line_400

    if UPDATE_IF_EXISTS:
        existing = RDK.Item(name, ITEM_TYPE_TARGET)
        if existing.Valid():
            existing.setAsCartesianTarget()
            existing.setPose(Ti)
            continue

    tgt = RDK.AddTarget(name, parent)
    tgt.setAsCartesianTarget()
    tgt.setPose(Ti)

print("Gotovo: napravljeno/azurirano targeta:", NPTS, f"({PREFIX}{START_NUM:03d}..{PREFIX}{(START_NUM+NPTS-1):03d})")

--- Python program Line_Following ---
from robodk.robolink import *
from robodk.robomath import *
import time

RDK = Robolink()

ROBOT2_NAME = 'Robot2'
PROG1_NAME  = 'Program_R1'

DT = 0.003
HOLD_TICKS = 6

# LOCK J4: 0.0 = hard lock (točno), stavi npr. 2.0 ako želiš malo tolerancije
J4_LOCK_TOL = 0.0

robot2 = RDK.Item(ROBOT2_NAME, ITEM_TYPE_ROBOT)
prog1  = RDK.Item(PROG1_NAME, ITEM_TYPE_PROGRAM)

if not robot2.Valid(): raise Exception("Robot2 nije pronađen")
if not prog1.Valid():  raise Exception("Program_R1 nije pronađen")

# targets
targets = []
t0 = RDK.Item('Start_Robot2', ITEM_TYPE_TARGET)
if not t0.Valid(): raise Exception("Nema targeta 'Start_Robot2'")
targets.append(t0)

for i in range(1, 401):
    ti = RDK.Item(f"Line_{i:03d}", ITEM_TYPE_TARGET)
    if not ti.Valid():
        raise Exception(f"Nedostaje Line_{i:03d}")
    targets.append(ti)

print("Ukupno targeta:", len(targets))

# brzine
robot2.setSpeed(1200)
robot2.setAcceleration(5000)
robot2.setSpeedJoints(300)
robot2.setAccelerationJoints(900)

# TMP target (fallback)
tmp = RDK.Item('TMP_R1', ITEM_TYPE_TARGET)
if not tmp.Valid():
    tmp = RDK.AddTarget('TMP_R1')
tmp.setAsCartesianTarget()

# joints helper
def fnum(v):
    while isinstance(v, (list, tuple)):
        if len(v) == 0: return None
        v = v[0]
    try:
        return float(v)
    except:
        s = str(v).replace('[','').replace(']','').strip()
        try: return float(s)
        except: return None

def joints6(j):
    try:
        out = [fnum(j[i]) for i in range(6)]
        if any(v is None for v in out): return None
        return out
    except:
        return None

def ang_diff(a, b):
    return (a - b + 180.0) % 360.0 - 180.0

def clamp(val, center, tol):
    if tol <= 0.0:
        return center
    d = ang_diff(val, center)
    if d > tol:  return center + tol
    if d < -tol: return center - tol
    return center + d

# frame/tool za IK
T_frame = robot2.PoseFrame()
T_tool  = robot2.PoseTool()

# idi na Pocetak (XYZ + rotacija)
T_abs0 = targets[0].PoseAbs()
tmp.setPoseAbs(T_abs0)
robot2.MoveJ(tmp, blocking=True)

# start jointovi (za lock J4 + seed za IK)
j_start = joints6(robot2.Joints())
if j_start is None:
    raise Exception("Ne mogu očitati start jointove Robot2")

j_prev = j_start[:]

# start Robot1
prog1.RunProgram()
print("START: prati XYZ+ROT, LOCK samo J4")

t_next = time.time()
idx = 0
tick_in_point = 0

while prog1.Busy() and idx < len(targets):

    now = time.time()
    if now < t_next:
        time.sleep(t_next - now)
    t_next += DT

    # uzmi CIJELI target pose (XYZ + ROT)
    T_abs = targets[idx].PoseAbs()

    ok = False
    try:
        T = invH(T_frame) * T_abs * invH(T_tool)
        j_sol = robot2.SolveIK(T, j_prev)
        j_new = joints6(j_sol)
        if j_new is not None:
            # LOCK J4 (index 3)
            j_new[3] = clamp(j_new[3], j_start[3], J4_LOCK_TOL)

            robot2.setJoints(j_new)
            j_prev = j_new
            ok = True
    except:
        ok = False

    if not ok:
        # fallback: MoveJ na pozu targeta
        tmp.setPoseAbs(T_abs)
        robot2.MoveJ(tmp, blocking=False)

    tick_in_point += 1
    if tick_in_point >= HOLD_TICKS:
        tick_in_point = 0
        idx += 1

# --- DODANO: zaustavi R1 kad se Robot2 zaustavi (tj. kad završi ova petlja) ---
if prog1.Busy():
    try:
        prog1.Stop()
    except:
        pass
    try:
        prog1.WaitFinished()
    except:
        pass
# ------------------------------------------------------------------------------

print("KRAJ.")

--- Python program Line_Following_konfg ---
from robodk.robolink import *
from robodk.robomath import *
import time
import csv
import os

RDK = Robolink()

ROBOT1_NAME = 'Robot1'
ROBOT2_NAME = 'Robot2'
PROG1_NAME  = 'Program_R1'

# =========================================================
# PODESAVANJA
# =========================================================
CONTROL_DT = 0.003
TARGET_HOLD_TICKS = 5
LOG_EVERY_N_TICKS = 1
J4_LOCK_TOL = 0.0

RESET_PAUSE_S = 0.2
# =========================================================

# -------- Items --------
robot1 = RDK.Item(ROBOT1_NAME, ITEM_TYPE_ROBOT)
robot2 = RDK.Item(ROBOT2_NAME, ITEM_TYPE_ROBOT)
prog1  = RDK.Item(PROG1_NAME, ITEM_TYPE_PROGRAM)

if not robot1.Valid(): raise Exception("Robot1 nije pronađen")
if not robot2.Valid(): raise Exception("Robot2 nije pronađen")
if not prog1.Valid():  raise Exception("Program_R1 nije pronađen")

t_start_r1 = RDK.Item('Start_Robot1', ITEM_TYPE_TARGET)
t_start_r2 = RDK.Item('Start_Robot2', ITEM_TYPE_TARGET)

if not t_start_r1.Valid(): raise Exception("Nema targeta 'Start_Robot1'")
if not t_start_r2.Valid(): raise Exception("Nema targeta 'Start_Robot2'")

# targets
targets = [t_start_r2]
for i in range(1, 401):
    ti = RDK.Item(f"Line_{i:03d}", ITEM_TYPE_TARGET)
    if not ti.Valid():
        raise Exception(f"Nedostaje Line_{i:03d}")
    targets.append(ti)

print("Ukupno targeta:", len(targets))

# brzine
robot2.setSpeed(1200)
robot2.setAcceleration(5000)
robot2.setSpeedJoints(300)
robot2.setAccelerationJoints(900)

# -------- helpers --------
def fnum(v):
    while isinstance(v, (list, tuple)):
        if len(v) == 0:
            return None
        v = v[0]
    try:
        return float(v)
    except:
        s = str(v).replace('[', '').replace(']', '').strip()
        try:
            return float(s)
        except:
            return None

def joints6(j):
    try:
        out = [fnum(j[i]) for i in range(6)]
        if any(v is None for v in out):
            return None
        return out
    except:
        return None

def ang_diff(a, b):
    return (a - b + 180.0) % 360.0 - 180.0

def clamp(val, center, tol):
    if tol <= 0.0:
        return center
    d = ang_diff(val, center)
    if d > tol:
        return center + tol
    if d < -tol:
        return center - tol
    return center + d

def stop_all_soft():
    try: prog1.Stop()
    except: pass
    try: robot1.Stop()
    except: pass
    try: robot2.Stop()
    except: pass

def find_tmp_list():
    # Trazi TMP_R1, TMP_R2, TMP_R3...
    out = []
    i = 1
    while True:
        it = RDK.Item(f"TMP_R{i}", ITEM_TYPE_TARGET)
        if not it.Valid():
            break
        it.setAsCartesianTarget()  # sigurnost
        out.append(it)
        i += 1
    return out

# -------- CSV --------
station_path = RDK.getParam('PATH_OPENSTATION')

# novo ime da ako je stari CSV otvoren u Excelu
out_file = os.path.join(station_path, "configs_line_following_detailed_notime.csv") if station_path else "configs_line_following_detailed_notime.csv"

csv_file = open(out_file, mode='w', newline='', encoding='utf-8')
writer = csv.writer(csv_file, delimiter=';')

#
writer.writerow([
    "config_idx","tmp_name",
    "sample_idx",
    "target_name","target_idx",
    "ik_ok",
    "r1_j1","r1_j2","r1_j3","r1_j4","r1_j5","r1_j6",
    "r2_j1","r2_j2","r2_j3","r2_j4","r2_j5","r2_j6"
])

tmp_list = find_tmp_list()
if len(tmp_list) == 0:
    csv_file.close()
    raise Exception("Nema TMP_R1/TMP_R2/... targeta u stanici.")

print("TMP targeti:", [t.Name() for t in tmp_list])

# -------- Run one config--------
def run_one_config(cfg_idx, tmp):
    print(f"\n=== CONFIG {cfg_idx}/{len(tmp_list)} using {tmp.Name()} ===")

    # ---------------------------------------------------------
    # RUCNI POSTUPAK (automatiziran)
    # 1) Start_Robot1
    # 2) Start_Robot2 preko AKTUALNOG TMP_Ri
    # 3) Pokreni line following
    # ---------------------------------------------------------
    stop_all_soft()
    time.sleep(RESET_PAUSE_S)

    # 1) Start_Robot1
    robot1.MoveJ(t_start_r1, blocking=True)

    # 2) Start_Robot2 preko bas tog TMP_Ri
    T_abs0 = t_start_r2.PoseAbs()
    tmp.setPoseAbs(T_abs0)
    robot2.MoveJ(tmp, blocking=True)

    # frame/tool (kao u tvom kodu)
    T_frame = robot2.PoseFrame()
    T_tool  = robot2.PoseTool()

    # idi na Pocetak (XYZ + rotacija)
    T_abs0 = targets[0].PoseAbs()
    tmp.setPoseAbs(T_abs0)
    robot2.MoveJ(tmp, blocking=True)

    # start jointovi (za lock J4 + seed za IK)
    j_start = joints6(robot2.Joints())
    if j_start is None:
        raise Exception("Ne mogu očitati start jointove Robot2")

    j_prev = j_start[:]

    # start Robot1
    prog1.RunProgram()
    print("START: prati XYZ+ROT, LOCK samo J4")

    t_next = time.time()
    idx = 0
    hold_tick = 0
    sample_idx = 0

    while prog1.Busy() and idx < len(targets):
        now = time.time()
        if now < t_next:
            time.sleep(t_next - now)
        t_next += CONTROL_DT

        # uzmi cijeli target pose (XYZ + ROT)
        T_abs = targets[idx].PoseAbs()

        ik_ok = 0
        try:
            T = invH(T_frame) * T_abs * invH(T_tool)
            j_sol = robot2.SolveIK(T, j_prev)
            j_new = joints6(j_sol)

            if j_new is not None:
                #
                j_new[3] = clamp(j_new[3], j_start[3], J4_LOCK_TOL)

                robot2.setJoints(j_new)
                j_prev = j_new
                ik_ok = 1
            else:
                #
                tmp.setPoseAbs(T_abs)
                robot2.MoveJ(tmp, blocking=False)
                ik_ok = 0
        except:
            try:
                tmp.setPoseAbs(T_abs)
                robot2.MoveJ(tmp, blocking=False)
            except:
                pass
            ik_ok = 0

        #LOG
        if (sample_idx % LOG_EVERY_N_TICKS) == 0:
            j1 = joints6(robot1.Joints()) or [""]*6
            j2 = joints6(robot2.Joints()) or [""]*6
            writer.writerow([
                cfg_idx, tmp.Name(),
                sample_idx,
                targets[idx].Name(), idx,
                ik_ok,
                *j1,
                *j2
            ])
            csv_file.flush()

        sample_idx += 1

        # target advance (brzina prolaska kroz targete)
        hold_tick += 1
        if hold_tick >= TARGET_HOLD_TICKS:
            hold_tick = 0
            idx += 1

    # Zaustavi R1 kad Robot2 zavrsi
    if prog1.Busy():
        try:
            prog1.Stop()
        except:
            pass
        try:
            prog1.WaitFinished()
        except:
            pass

    stop_all_soft()

# -------- Main loop: TMP_R1, TMP_R2, TMP_R3... --------
for i, tmp_i in enumerate(tmp_list, start=1):
    try:
        run_one_config(i, tmp_i)
    except Exception as e:
        print("EXCEPTION:", str(e))
        stop_all_soft()
        time.sleep(RESET_PAUSE_S)
        continue

csv_file.close()
print("\nSpremljeno:", out_file)
print("KRAJ.")

--- Python program Line_Following_Analiza ---
import csv
import os
import math

# =========================================================
# PODESI PUTANJU DO TVOG SNIMLJENOG CSV-a
# =========================================================
INPUT_CSV = r"C:/Users/xgami/Downloads/Završni_Stanice_Ispravak/Završni_Stanice_Ispravak/configs_line_following_detailed_notime.csv"

# Pragovi za detekciju "reset" / naglih skokova
RESET_JUMP_ANY_DEG   = 120.0   # ako bilo koji joint skoci vise od ovoga
RESET_JUMP_TOTAL_DEG = 260.0   # ili ako zbroj svih skokova prede ovo



def ang_diff(a, b):
    """Kutna razlika uz wrap (-180..180)."""
    return (a - b + 180.0) % 360.0 - 180.0


def ffloat(x, default=None):
    try:
        return float(str(x).strip().replace(",", "."))
    except:
        return default


def fint(x, default=None):
    try:
        return int(float(str(x).strip()))
    except:
        return default


def percentile(values, p):
    if not values:
        return 0.0
    vals = sorted(values)
    if len(vals) == 1:
        return vals[0]
    k = (len(vals) - 1) * (p / 100.0)
    f = int(math.floor(k))
    c = int(math.ceil(k))
    if f == c:
        return vals[f]
    d0 = vals[f] * (c - k)
    d1 = vals[c] * (k - f)
    return d0 + d1


def read_samples(path):
    if not os.path.isfile(path):
        raise FileNotFoundError("Ne mogu naći ulazni CSV: " + path)

    rows = []
    with open(path, "r", encoding="utf-8", newline="") as f:
        reader = csv.DictReader(f, delimiter=';')
        if reader.fieldnames is None:
            raise Exception("CSV nema header.")

        for r in reader:
            if not r:
                continue
            if r.get("config_idx", "").strip() == "":
                continue
            if r.get("r2_j1", "").strip() == "":
                continue

            cfg_idx = fint(r.get("config_idx"))
            sample_idx = fint(r.get("sample_idx"), 0)
            ik_ok = fint(r.get("ik_ok"), 0)

            if cfg_idx is None:
                continue

            r1 = [ffloat(r.get(f"r1_j{i}"), 0.0) for i in range(1, 7)]
            r2 = [ffloat(r.get(f"r2_j{i}"), 0.0) for i in range(1, 7)]

            if any(v is None for v in r1 + r2):
                continue

            rows.append({
                "config_idx": cfg_idx,
                "tmp_name": (r.get("tmp_name") or "").strip(),
                "sample_idx": sample_idx,
                "target_name": (r.get("target_name") or "").strip(),
                "target_idx": fint(r.get("target_idx"), 0),
                "ik_ok": ik_ok,
                "r1": r1,
                "r2": r2,
                "raw": r
            })

    if len(rows) == 0:
        raise Exception("CSV je pročitan, ali nema valjanih redova podataka.")

    return rows


def group_by_config(rows):
    groups = {}
    for row in rows:
        key = (row["config_idx"], row["tmp_name"])
        if key not in groups:
            groups[key] = []
        groups[key].append(row)

    # Sort po sample_idx (za replay i analizu skokova)
    for key in groups:
        groups[key].sort(key=lambda x: x["sample_idx"])
    return groups


def analyze_group(samples):
    ik_fail_count = 0
    jumps_any = []
    jumps_total = []
    reset_events = 0

    for s in samples:
        if s["ik_ok"] != 1:
            ik_fail_count += 1

    for i in range(1, len(samples)):
        prev_q = samples[i - 1]["r2"]
        curr_q = samples[i]["r2"]

        dj = [abs(ang_diff(curr_q[j], prev_q[j])) for j in range(6)]
        max_jump = max(dj)
        total_jump = sum(dj)

        jumps_any.append(max_jump)
        jumps_total.append(total_jump)

        if (max_jump >= RESET_JUMP_ANY_DEG) or (total_jump >= RESET_JUMP_TOTAL_DEG):
            reset_events += 1

    max_joint_jump = max(jumps_any) if jumps_any else 0.0
    max_total_jump = max(jumps_total) if jumps_total else 0.0
    p95_total = percentile(jumps_total, 95) if jumps_total else 0.0
    avg_total = (sum(jumps_total) / len(jumps_total)) if jumps_total else 0.0

    # Score: ogromna kazna na reset, pa IK fail, pa skokovi
    score = (
        reset_events * 1_000_000.0 +
        ik_fail_count * 10_000.0 +
        max_total_jump * 100.0 +
        p95_total * 10.0 +
        avg_total
    )

    return {
        "samples": len(samples),
        "reset_events": reset_events,
        "ik_fail_count": ik_fail_count,
        "max_joint_jump_deg": round(max_joint_jump, 4),
        "max_total_jump_deg": round(max_total_jump, 4),
        "p95_total_jump_deg": round(p95_total, 4),
        "avg_total_jump_deg": round(avg_total, 4),
        "score": round(score, 4),
    }


def safe_write_csv(path, header, rows):
    # Ako je file otvoren u Excelu -> fallback ime
    try_paths = [path]
    base, ext = os.path.splitext(path)
    try_paths.append(base + "_new" + ext)
    try_paths.append(base + "_out" + ext)

    last_err = None
    for p in try_paths:
        try:
            with open(p, "w", encoding="utf-8", newline="") as f:
                w = csv.writer(f, delimiter=';')
                w.writerow(header)
                for row in rows:
                    w.writerow(row)
            return p
        except PermissionError as e:
            last_err = e
            continue

    raise last_err if last_err else Exception("Ne mogu zapisati CSV.")


def main():
    rows = read_samples(INPUT_CSV)
    groups = group_by_config(rows)

    if len(groups) == 0:
        raise Exception("Nema grupa konfiguracija za analizu.")

    summary = []
    best_key = None
    best_metrics = None
    best_score = None

    for (cfg_idx, tmp_name), samples in sorted(groups.items(), key=lambda x: x[0][0]):
        m = analyze_group(samples)
        rec = {
            "config_idx": cfg_idx,
            "tmp_name": tmp_name,
            **m
        }
        summary.append(rec)

        if (best_score is None) or (m["score"] < best_score):
            best_score = m["score"]
            best_key = (cfg_idx, tmp_name)
            best_metrics = m

    # Folder outputa = isti folder gdje je input CSV
    out_dir = os.path.dirname(INPUT_CSV) if os.path.dirname(INPUT_CSV) else "."

    # 1) Summary CSV
    summary_header = [
        "config_idx", "tmp_name",
        "samples", "reset_events", "ik_fail_count",
        "max_joint_jump_deg", "max_total_jump_deg",
        "p95_total_jump_deg", "avg_total_jump_deg",
        "score"
    ]
    summary_rows = []
    for s in summary:
        summary_rows.append([
            s["config_idx"], s["tmp_name"],
            s["samples"], s["reset_events"], s["ik_fail_count"],
            s["max_joint_jump_deg"], s["max_total_jump_deg"],
            s["p95_total_jump_deg"], s["avg_total_jump_deg"],
            s["score"]
        ])

    summary_path = safe_write_csv(
        os.path.join(out_dir, "analysis_summary.csv"),
        summary_header,
        summary_rows
    )

    # 2) Best config only CSV (isti header kao original!)
    best_samples = groups[best_key]

    # Uzmi original header iz prvog raw reda
    raw_header = list(best_samples[0]["raw"].keys())

    best_rows = []
    for s in best_samples:
        best_rows.append([s["raw"].get(h, "") for h in raw_header])

    best_path = safe_write_csv(
        os.path.join(out_dir, "best_config_only.csv"),
        raw_header,
        best_rows
    )

    # Print rezultat
    print("\n================ REZULTAT ================")
    print("Najbolja konfiguracija:")
    print("  config_idx:", best_key[0])
    print("  tmp_name:", best_key[1])
    print("  samples:", best_metrics["samples"])
    print("  reset_events:", best_metrics["reset_events"])
    print("  ik_fail_count:", best_metrics["ik_fail_count"])
    print("  max_joint_jump_deg:", best_metrics["max_joint_jump_deg"])
    print("  max_total_jump_deg:", best_metrics["max_total_jump_deg"])
    print("  p95_total_jump_deg:", best_metrics["p95_total_jump_deg"])
    print("  avg_total_jump_deg:", best_metrics["avg_total_jump_deg"])
    print("  score:", best_metrics["score"])
    print("==========================================")

    print("\nSpremljeno:")
    print("  Summary :", summary_path)
    print("  Best CSV:", best_path)
    print("\nReplay koristi ovaj file -> best_config_only.csv")

